    |   movel([-0.157173, -0.854007, -2.792927, -1.065455, 1.570796, 1.413623],accel_mss,speed_ms,0,blend_radius_m)
    |   movel([-0.155636, -0.852773, -2.793167, -1.066449, 1.570796, 1.415161],accel_mss,speed_ms,0,blend_radius_m)
    |   movel([-0.153982, -0.851875, -2.793341, -1.067172, 1.570796, 1.416814],accel_mss,speed_ms,0,blend_radius_m)
    |   movel([-0.150724, -0.850900, -2.793530, -1.067959, 1.570796, 1.420072],accel_mss,speed_ms,0,blend_radius_m)
    |   movel([-0.148143, -0.850668, -2.793575, -1.068146, 1.570796, 1.422653],accel_mss,speed_ms,0,blend_radius_m)
    |   movel([-0.149321, -0.848135, -2.794062, -1.070192, 1.570796, 1.421476],accel_mss,speed_ms,0,blend_radius_m)
    |   movel([-0.151025, -0.846251, -2.794422, -1.071716, 1.570796, 1.419772],accel_mss,speed_ms,0,blend_radius_m)
    |   movel([-0.155392, -0.843635, -2.794919, -1.073835, 1.570796, 1.415404],accel_mss,speed_ms,0,blend_radius_m)
    |   movel([-0.159988, -0.841179, -2.795382, -1.075828, 1.570796, 1.410808],accel_mss,speed_ms,0,blend_radius_m)
    |   movel([-0.161984, -0.839490, -2.795698, -1.077201, 1.570796, 1.408813],accel_mss,speed_ms,0,blend_radius_m)
    |   movel([-0.163557, -0.837206, -2.796124, -1.079060, 1.570796, 1.407239],accel_mss,speed_ms,0,blend_radius_m)
    |   movel([-0.164261, -0.835458, -2.796447, -1.080484, 1.570796, 1.406535],accel_mss,speed_ms,0,blend_radius_m)
    |   movel([-0.164602, -0.833827, -2.796748, -1.081815, 1.570796, 1.406195],accel_mss,speed_ms,0,blend_radius_m)
    |   movel([-0.164612, -0.832318, -2.797024, -1.083047, 1.570796, 1.406184],accel_mss,speed_ms,0,blend_radius_m)
    |   movel([-0.164323, -0.830942, -2.797275, -1.084171, 1.570796, 1.406473],accel_mss,speed_ms,0,blend_radius_m)
    |   movel([-0.163779, -0.829715, -2.797499, -1.085176, 1.570796, 1.407017],accel_mss,speed_ms,0,blend_radius_m)
    |   movel([-0.163009, -0.828631, -2.797695, -1.086063, 1.570796, 1.407787],accel_mss,speed_ms,0,blend_radius_m)
    |   movel([-0.162059, -0.827711, -2.797861, -1.086817, 1.570796, 1.408737],accel_mss,speed_ms,0,blend_radius_m)
    |   movel([-0.160956, -0.826959, -2.797997, -1.087433, 1.570796, 1.409840],accel_mss,speed_ms,0,blend_radius_m)
    |   movel([-0.159743, -0.826388, -2.798099, -1.087901, 1.570796, 1.411053],accel_mss,speed_ms,0,blend_radius_m)
    |   movel([-0.158463, -0.826010, -2.798167, -1.088211, 1.570796, 1.412333],accel_mss,speed_ms,0,blend_radius_m)
    |   movel([-0.155834, -0.825858, -2.798195, -1.088336, 1.570796, 1.414963],accel_mss,speed_ms,0,blend_radius_m)
    |   movel([-0.153372, -0.826573, -2.798066, -1.087750, 1.570796, 1.417424],accel_mss,speed_ms,0,blend_radius_m)
    |   movel([-0.151377, -0.828225, -2.797768, -1.086396, 1.570796, 1.419420],accel_mss,speed_ms,0,blend_radius_m)
    |   movel([-0.151142, -0.825056, -2.798338, -1.088994, 1.570796, 1.419654],accel_mss,speed_ms,0,blend_radius_m)
    |   movel([-0.151297, -0.822338, -2.798823, -1.091228, 1.570796, 1.419499],accel_mss,speed_ms,0,blend_radius_m)
    |   movel([-0.151760, -0.819974, -2.799241, -1.093173, 1.570796, 1.419036],accel_mss,speed_ms,0,blend_radius_m)
    |   movel([-0.154101, -0.813819, -2.800316, -1.098253, 1.570796, 1.416695],accel_mss,speed_ms,0,blend_radius_m)
    |   movel([-0.155566, -0.809336, -2.801087, -1.101966, 1.570796, 1.415230],accel_mss,speed_ms,0,blend_radius_m)
    |   movel([-0.155893, -0.807231, -2.801445, -1.103713, 1.570796, 1.414904],accel_mss,speed_ms,0,blend_radius_m)
    |   movel([-0.155922, -0.805199, -2.801789, -1.105401, 1.570796, 1.414875],accel_mss,speed_ms,0,blend_radius_m)
    |   movel([-0.155690, -0.803274, -2.802112, -1.107003, 1.570796, 1.415106],accel_mss,speed_ms,0,blend_radius_m)
    |   movel([-0.155226, -0.801477, -2.802413, -1.108500, 1.570796, 1.415570],accel_mss,speed_ms,0,blend_radius_m)
    |   movel([-0.154569, -0.799836, -2.802685, -1.109868, 1.570796, 1.416227],accel_mss,speed_ms,0,blend_radius_m)
    |   movel([-0.153748, -0.798375, -2.802927, -1.111087, 1.570796, 1.417049],accel_mss,speed_ms,0,blend_radius_m)
    |   movel([-0.152797, -0.797121, -2.803133, -1.112135, 1.570796, 1.417999],accel_mss,speed_ms,0,blend_radius_m)
    |   movel([-0.151752, -0.796103, -2.803301, -1.112985, 1.570796, 1.419044],accel_mss,speed_ms,0,blend_radius_m)
    |   movel([-0.150649, -0.795350, -2.803424, -1.113616, 1.570796, 1.420147],accel_mss,speed_ms,0,blend_radius_m)
    |   movel([-0.149524, -0.794885, -2.803500, -1.114004, 1.570796, 1.421272],accel_mss,speed_ms,0,blend_radius_m)
    |   movel([-0.148407, -0.794733, -2.803525, -1.114131, 1.570796, 1.422389],accel_mss,speed_ms,0,blend_radius_m)
    |   movel([-0.147335, -0.794925, -2.803493, -1.113970, 1.570796, 1.423462],accel_mss,speed_ms,0,blend_radius_m)
    |   movel([-0.146348, -0.795490, -2.803401, -1.113498, 1.570796, 1.424449],accel_mss,speed_ms,0,blend_radius_m)
    |   movel([-0.145476, -0.796449, -2.803244, -1.112696, 1.570796, 1.425320],accel_mss,speed_ms,0,blend_radius_m)
    |   movel([-0.144756, -0.797829, -2.803017, -1.111543, 1.570796, 1.426040],accel_mss,speed_ms,0,blend_radius_m)
    |   movel([-0.144218, -0.799645, -2.802717, -1.110027, 1.570796, 1.426578],accel_mss,speed_ms,0,blend_radius_m)
    |   movel([-0.142768, -0.796226, -2.803280, -1.112882, 1.570796, 1.428028],accel_mss,speed_ms,0,blend_radius_m)
    |   movel([-0.141654, -0.792950, -2.803815, -1.115625, 1.570796, 1.429142],accel_mss,speed_ms,0,blend_radius_m)
    |   movel([-0.140811, -0.789788, -2.804325, -1.118275, 1.570796, 1.429985],accel_mss,speed_ms,0,blend_radius_m)
    |   movel([-0.140168, -0.786710, -2.804817, -1.120861, 1.570796, 1.430628],accel_mss,speed_ms,0,blend_radius_m)
    |   movel([-0.138139, -0.774609, -2.806707, -1.131074, 1.570796, 1.432657],accel_mss,speed_ms,0,blend_radius_m)
    |   movel([-0.137268, -0.770063, -2.807398, -1.134928, 1.570796, 1.433528],accel_mss,speed_ms,0,blend_radius_m)
    |   movel([-0.135786, -0.764437, -2.808239, -1.139713, 1.570796, 1.435010],accel_mss,speed_ms,0,blend_radius_m)
    |   movel([-0.134635, -0.761547, -2.808665, -1.142177, 1.570796, 1.436162],accel_mss,speed_ms,0,blend_radius_m)
    |   movel([-0.133113, -0.758786, -2.809068, -1.144534, 1.570796, 1.437684],accel_mss,speed_ms,0,blend_radius_m)
    |   movel([-0.132184, -0.757494, -2.809256, -1.145639, 1.570796, 1.438613],accel_mss,speed_ms,0,blend_radius_m)
    |   movel([-0.129965, -0.755171, -2.809591, -1.147627, 1.570796, 1.440832],accel_mss,speed_ms,0,blend_radius_m)
    |   movel([-0.128651, -0.754181, -2.809733, -1.148475, 1.570796, 1.442146],accel_mss,speed_ms,0,blend_radius_m)
    |   movel([-0.127337, -0.753612, -2.809815, -1.148962, 1.570796, 1.443459],accel_mss,speed_ms,0,blend_radius_m)
    |   movel([-0.126342, -0.753754, -2.809794, -1.148841, 1.570796, 1.444454],accel_mss,speed_ms,0,blend_radius_m)
    |   movel([-0.125121, -0.755288, -2.809574, -1.147527, 1.570796, 1.445675],accel_mss,speed_ms,0,blend_radius_m)
    |   movel([-0.124184, -0.758153, -2.809161, -1.145076, 1.570796, 1.446612],accel_mss,speed_ms,0,blend_radius_m)
    |   movel([-0.123601, -0.761345, -2.808695, -1.142350, 1.570796, 1.447196],accel_mss,speed_ms,0,blend_radius_m)
    |   movel([-0.121151, -0.756396, -2.809415, -1.146579, 1.570796, 1.449645],accel_mss,speed_ms,0,blend_radius_m)
    |   movel([-0.118326, -0.751367, -2.810134, -1.150887, 1.570796, 1.452470],accel_mss,speed_ms,0,blend_radius_m)
    |   movel([-0.115181, -0.746327, -2.810844, -1.155218, 1.570796, 1.455615],accel_mss,speed_ms,0,blend_radius_m)
    |   movel([-0.111786, -0.741349, -2.811533, -1.159508, 1.570796, 1.459011],accel_mss,speed_ms,0,blend_radius_m)
    |   movel([-0.104952, -0.731339, -2.812883, -1.168167, 1.570796, 1.465845],accel_mss,speed_ms,0,blend_radius_m)
    |   movel([-0.102905, -0.728573, -2.813248, -1.170568, 1.570796, 1.467892],accel_mss,speed_ms,0,blend_radius_m)
    |   movel([-0.100882, -0.726090, -2.813573, -1.172726, 1.570796, 1.469915],accel_mss,speed_ms,0,blend_radius_m)
    |   movel([-0.098956, -0.724081, -2.813833, -1.174475, 1.570796, 1.471840],accel_mss,speed_ms,0,blend_radius_m)
    |   movel([-0.097220, -0.722741, -2.814006, -1.175641, 1.570796, 1.473576],accel_mss,speed_ms,0,blend_radius_m)
    |   movel([-0.095733, -0.722296, -2.814064, -1.176030, 1.570796, 1.475063],accel_mss,speed_ms,0,blend_radius_m)
    |   movel([-0.094670, -0.722789, -2.814000, -1.175600, 1.570796, 1.476126],accel_mss,speed_ms,0,blend_radius_m)
    |   movel([-0.094003, -0.724018, -2.813842, -1.174529, 1.570796, 1.476793],accel_mss,speed_ms,0,blend_radius_m)
    |   movel([-0.093720, -0.725788, -2.813612, -1.172989, 1.570796, 1.477077],accel_mss,speed_ms,0,blend_radius_m)
    |   movel([-0.093794, -0.727894, -2.813337, -1.171158, 1.570796, 1.477002],accel_mss,speed_ms,0,blend_radius_m)
    |   movel([-0.094201, -0.730131, -2.813043, -1.169215, 1.570796, 1.476595],accel_mss,speed_ms,0,blend_radius_m)
    |   movel([-0.094921, -0.732302, -2.812755, -1.167332, 1.570796, 1.475876],accel_mss,speed_ms,0,blend_radius_m)
    |   movel([-0.095934, -0.734211, -2.812500, -1.165677, 1.570796, 1.474862],accel_mss,speed_ms,0,blend_radius_m)
    |   movel([-0.089576, -0.725324, -2.813672, -1.173393, 1.570796, 1.481220],accel_mss,speed_ms,0,blend_radius_m)
    |   movel([-0.086162, -0.720979, -2.814232, -1.177177, 1.570796, 1.484634],accel_mss,speed_ms,0,blend_radius_m)
    |   movel([-0.082605, -0.716751, -2.814769, -1.180869, 1.570796, 1.488191],accel_mss,speed_ms,0,blend_radius_m)
    |   movel([-0.078927, -0.712679, -2.815278, -1.184431, 1.570796, 1.491869],accel_mss,speed_ms,0,blend_radius_m)
    |   movel([-0.075137, -0.708803, -2.815756, -1.187829, 1.570796, 1.495659],accel_mss,speed_ms,0,blend_radius_m)
    |   movel([-0.071252, -0.705165, -2.816199, -1.191025, 1.570796, 1.499544],accel_mss,speed_ms,0,blend_radius_m)
    |   movel([-0.067291, -0.701802, -2.816603, -1.193984, 1.570796, 1.503506],accel_mss,speed_ms,0,blend_radius_m)
    |   movel([-0.064593, -0.700056, -2.816811, -1.195522, 1.570796, 1.506203],accel_mss,speed_ms,0,blend_radius_m)
    |   movel([-0.061701, -0.698911, -2.816946, -1.196532, 1.570796, 1.509095],accel_mss,speed_ms,0,blend_radius_m)
    |   movel([-0.060444, -0.698737, -2.816967, -1.196685, 1.570796, 1.510352],accel_mss,speed_ms,0,blend_radius_m)
    |   movel([-0.059448, -0.698913, -2.816946, -1.196530, 1.570796, 1.511348],accel_mss,speed_ms,0,blend_radius_m)
    |   movel([-0.058813, -0.699508, -2.816876, -1.196006, 1.570796, 1.511984],accel_mss,speed_ms,0,blend_radius_m)
    |   movel([-0.058648, -0.700593, -2.816747, -1.195049, 1.570796, 1.512148],accel_mss,speed_ms,0,blend_radius_m)
    |   movel([-0.059026, -0.702035, -2.816575, -1.193779, 1.570796, 1.511771],accel_mss,speed_ms,0,blend_radius_m)
    |   movel([-0.059804, -0.703666, -2.816380, -1.192343, 1.570796, 1.510992],accel_mss,speed_ms,0,blend_radius_m)
    |   movel([-0.062125, -0.707350, -2.815934, -1.189105, 1.570796, 1.508671],accel_mss,speed_ms,0,blend_radius_m)
    |   movel([-0.064902, -0.710819, -2.815509, -1.186061, 1.570796, 1.505895],accel_mss,speed_ms,0,blend_radius_m)
    |   movel([-0.067942, -0.714038, -2.815109, -1.183242, 1.570796, 1.502854],accel_mss,speed_ms,0,blend_radius_m)
    |   movel([-0.071057, -0.716970, -2.814741, -1.180677, 1.570796, 1.499740],accel_mss,speed_ms,0,blend_radius_m)
    |   movel([-0.067028, -0.715222, -2.814961, -1.182206, 1.570796, 1.503768],accel_mss,speed_ms,0,blend_radius_m)
    |   movel([-0.062835, -0.712992, -2.815240, -1.184158, 1.570796, 1.507961],accel_mss,speed_ms,0,blend_radius_m)
    |   movel([-0.058521, -0.710309, -2.815572, -1.186509, 1.570796, 1.512275],accel_mss,speed_ms,0,blend_radius_m)
    |   movel([-0.054124, -0.707195, -2.815953, -1.189242, 1.570796, 1.516672],accel_mss,speed_ms,0,blend_radius_m)
    |   movel([-0.050646, -0.704373, -2.816295, -1.191722, 1.570796, 1.520151],accel_mss,speed_ms,0,blend_radius_m)
    |   movel([-0.043815, -0.698292, -2.817019, -1.197078, 1.570796, 1.526981],accel_mss,speed_ms,0,blend_radius_m)
    |   movel([-0.040303, -0.695418, -2.817356, -1.199615, 1.570796, 1.530493],accel_mss,speed_ms,0,blend_radius_m)
    |   movel([-0.036299, -0.692430, -2.817703, -1.202257, 1.570796, 1.534498],accel_mss,speed_ms,0,blend_radius_m)
    |   movel([-0.029550, -0.687751, -2.818237, -1.206401, 1.570796, 1.541246],accel_mss,speed_ms,0,blend_radius_m)
    |   movel([-0.026322, -0.685794, -2.818458, -1.208137, 1.570796, 1.544475],accel_mss,speed_ms,0,blend_radius_m)
    |   movel([-0.023824, -0.684639, -2.818588, -1.209162, 1.570796, 1.546972],accel_mss,speed_ms,0,blend_radius_m)
    |   movel([-0.022997, -0.684488, -2.818605, -1.209296, 1.570796, 1.547799],accel_mss,speed_ms,0,blend_radius_m)
    |   movel([-0.022536, -0.684694, -2.818582, -1.209113, 1.570796, 1.548260],accel_mss,speed_ms,0,blend_radius_m)
    |   movel([-0.022492, -0.685295, -2.818514, -1.208579, 1.570796, 1.548305],accel_mss,speed_ms,0,blend_radius_m)
    |   movel([-0.022929, -0.686348, -2.818396, -1.207645, 1.570796, 1.547867],accel_mss,speed_ms,0,blend_radius_m)
    |   movel([-0.024592, -0.689011, -2.818094, -1.205283, 1.570796, 1.546204],accel_mss,speed_ms,0,blend_radius_m)
    |   movel([-0.026746, -0.691820, -2.817773, -1.202796, 1.570796, 1.544050],accel_mss,speed_ms,0,blend_radius_m)
    |   movel([-0.029251, -0.694704, -2.817439, -1.200246, 1.570796, 1.541546],accel_mss,speed_ms,0,blend_radius_m)
    |   movel([-0.031954, -0.697567, -2.817105, -1.197717, 1.570796, 1.538842],accel_mss,speed_ms,0,blend_radius_m)
    |   movel([-0.037413, -0.702922, -2.816469, -1.192998, 1.570796, 1.533384],accel_mss,speed_ms,0,blend_radius_m)
    |   movel([-0.041996, -0.707237, -2.815948, -1.189204, 1.570796, 1.528800],accel_mss,speed_ms,0,blend_radius_m)
    |   movel([-0.039684, -0.706721, -2.816010, -1.189657, 1.570796, 1.531113],accel_mss,speed_ms,0,blend_radius_m)
    |   movel([-0.037246, -0.705917, -2.816108, -1.190364, 1.570796, 1.533551],accel_mss,speed_ms,0,blend_radius_m)
    |   movel([-0.032075, -0.703597, -2.816388, -1.192404, 1.570796, 1.538721],accel_mss,speed_ms,0,blend_radius_m)
    |   movel([-0.026629, -0.700547, -2.816752, -1.195089, 1.570796, 1.544167],accel_mss,speed_ms,0,blend_radius_m)
    |   movel([-0.021050, -0.697047, -2.817166, -1.198176, 1.570796, 1.549746],accel_mss,speed_ms,0,blend_radius_m)
    |   movel([-0.016407, -0.693865, -2.817537, -1.200987, 1.570796, 1.554390],accel_mss,speed_ms,0,blend_radius_m)
    |   movel([-0.002304, -0.683687, -2.818694, -1.210008, 1.570796, 1.568493],accel_mss,speed_ms,0,blend_radius_m)
    |   movel([0.000307, -0.682237, -2.818856, -1.211296, 1.570796, 1.571103],accel_mss,speed_ms,0,blend_radius_m)
    |   movel([0.002343, -0.681707, -2.818914, -1.211768, 1.570796, 1.573139],accel_mss,speed_ms,0,blend_radius_m)
    |   movel([0.002760, -0.682018, -2.818880, -1.211491, 1.570796, 1.573556],accel_mss,speed_ms,0,blend_radius_m)
    |   movel([0.002568, -0.682838, -2.818789, -1.210762, 1.570796, 1.573364],accel_mss,speed_ms,0,blend_radius_m)
    |   movel([0.001613, -0.684258, -2.818631, -1.209501, 1.570796, 1.572410],accel_mss,speed_ms,0,blend_radius_m)
    |   movel([-0.000256, -0.686365, -2.818394, -1.207630, 1.570796, 1.570541],accel_mss,speed_ms,0,blend_radius_m)
    |   movel([-0.003382, -0.689438, -2.818046, -1.204905, 1.570796, 1.567415],accel_mss,speed_ms,0,blend_radius_m)
    |   movel([-0.006983, -0.692611, -2.817682, -1.202096, 1.570796, 1.563814],accel_mss,speed_ms,0,blend_radius_m)
    |   movel([-0.010526, -0.695305, -2.817369, -1.199714, 1.570796, 1.560271],accel_mss,speed_ms,0,blend_radius_m)
    |   movel([-0.012112, -0.696296, -2.817254, -1.198839, 1.570796, 1.558684],accel_mss,speed_ms,0,blend_radius_m)
    |   movel([-0.013481, -0.696943, -2.817178, -1.198268, 1.570796, 1.557315],accel_mss,speed_ms,0,blend_radius_m)
    |   movel([-0.008162, -0.696506, -2.817229, -1.198654, 1.570796, 1.562634],accel_mss,speed_ms,0,blend_radius_m)
    |   movel([-0.002460, -0.695324, -2.817367, -1.199698, 1.570796, 1.568336],accel_mss,speed_ms,0,blend_radius_m)
    |   movel([0.003547, -0.693539, -2.817574, -1.201275, 1.570796, 1.574343],accel_mss,speed_ms,0,blend_radius_m)
    |   movel([0.009790, -0.691297, -2.817833, -1.203259, 1.570796, 1.580586],accel_mss,speed_ms,0,blend_radius_m)
    |   movel([0.022658, -0.686000, -2.818435, -1.207954, 1.570796, 1.593454],accel_mss,speed_ms,0,blend_radius_m)
    |   movel([0.035476, -0.680608, -2.819036, -1.212745, 1.570796, 1.606273],accel_mss,speed_ms,0,blend_radius_m)
    |   movel([0.037595, -0.680073, -2.819095, -1.213222, 1.570796, 1.608391],accel_mss,speed_ms,0,blend_radius_m)
    |   movel([0.038280, -0.680335, -2.819066, -1.212988, 1.570796, 1.609077],accel_mss,speed_ms,0,blend_radius_m)
    |   movel([0.038454, -0.681179, -2.818973, -1.212237, 1.570796, 1.609251],accel_mss,speed_ms,0,blend_radius_m)
    |   movel([0.038045, -0.682450, -2.818832, -1.211107, 1.570796, 1.608841],accel_mss,speed_ms,0,blend_radius_m)
    |   movel([0.035891, -0.686011, -2.818434, -1.207944, 1.570796, 1.606687],accel_mss,speed_ms,0,blend_radius_m)
    |   movel([0.034360, -0.688066, -2.818202, -1.206121, 1.570796, 1.605157],accel_mss,speed_ms,0,blend_radius_m)
    |   movel([0.030931, -0.691910, -2.817763, -1.202716, 1.570796, 1.601727],accel_mss,speed_ms,0,blend_radius_m)
    |   movel([0.027173, -0.695360, -2.817363, -1.199666, 1.570796, 1.597970],accel_mss,speed_ms,0,blend_radius_m)
    |   movel([0.023244, -0.698409, -2.817005, -1.196974, 1.570796, 1.594040],accel_mss,speed_ms,0,blend_radius_m)
    |   movel([0.019315, -0.701027, -2.816695, -1.194667, 1.570796, 1.590111],accel_mss,speed_ms,0,blend_radius_m)
    |   movel([0.015548, -0.703199, -2.816436, -1.192754, 1.570796, 1.586344],accel_mss,speed_ms,0,blend_radius_m)
    |   movel([0.012105, -0.704898, -2.816231, -1.191260, 1.570796, 1.582901],accel_mss,speed_ms,0,blend_radius_m)
    |   movel([0.009158, -0.706089, -2.816087, -1.190213, 1.570796, 1.579955],accel_mss,speed_ms,0,blend_radius_m)
    |   movel([0.009122, -0.706976, -2.815979, -1.189433, 1.570796, 1.579918],accel_mss,speed_ms,0,blend_radius_m)
    |   movel([0.009634, -0.707378, -2.815930, -1.189081, 1.570796, 1.580430],accel_mss,speed_ms,0,blend_radius_m)
    |   movel([0.011224, -0.707724, -2.815888, -1.188777, 1.570796, 1.582020],accel_mss,speed_ms,0,blend_radius_m)
    |   movel([0.013030, -0.707717, -2.815889, -1.188783, 1.570796, 1.583826],accel_mss,speed_ms,0,blend_radius_m)
    |   movel([0.017003, -0.707079, -2.815967, -1.189343, 1.570796, 1.587799],accel_mss,speed_ms,0,blend_radius_m)
    |   movel([0.024091, -0.705495, -2.816159, -1.190735, 1.570796, 1.594887],accel_mss,speed_ms,0,blend_radius_m)
    |   movel([0.031302, -0.703602, -2.816387, -1.192399, 1.570796, 1.602098],accel_mss,speed_ms,0,blend_radius_m)
    |   movel([0.046101, -0.699018, -2.816934, -1.196438, 1.570796, 1.616897],accel_mss,speed_ms,0,blend_radius_m)
    |   movel([0.050206, -0.697835, -2.817073, -1.197481, 1.570796, 1.621002],accel_mss,speed_ms,0,blend_radius_m)
    |   movel([0.052798, -0.697331, -2.817132, -1.197926, 1.570796, 1.623594],accel_mss,speed_ms,0,blend_radius_m)
    |   movel([0.055274, -0.697154, -2.817153, -1.198082, 1.570796, 1.626070],accel_mss,speed_ms,0,blend_radius_m)
    |   movel([0.057259, -0.697513, -2.817111, -1.197765, 1.570796, 1.628055],accel_mss,speed_ms,0,blend_radius_m)
    |   movel([0.058392, -0.698596, -2.816983, -1.196809, 1.570796, 1.629188],accel_mss,speed_ms,0,blend_radius_m)
    |   movel([0.058534, -0.699464, -2.816881, -1.196044, 1.570796, 1.629331],accel_mss,speed_ms,0,blend_radius_m)
    |   movel([0.058333, -0.700583, -2.816748, -1.195058, 1.570796, 1.629130],accel_mss,speed_ms,0,blend_radius_m)
    |   movel([0.057737, -0.701985, -2.816581, -1.193823, 1.570796, 1.628533],accel_mss,speed_ms,0,blend_radius_m)
    |   movel([0.056715, -0.703679, -2.816378, -1.192332, 1.570796, 1.627511],accel_mss,speed_ms,0,blend_radius_m)
    |   movel([0.055222, -0.705253, -2.816188, -1.190947, 1.570796, 1.626018],accel_mss,speed_ms,0,blend_radius_m)
    |   movel([0.053193, -0.706766, -2.816005, -1.189618, 1.570796, 1.623989],accel_mss,speed_ms,0,blend_radius_m)
    |   movel([0.042343, -0.713656, -2.815157, -1.183576, 1.570796, 1.613139],accel_mss,speed_ms,0,blend_radius_m)
    |   movel([0.038709, -0.715494, -2.814927, -1.181968, 1.570796, 1.609506],accel_mss,speed_ms,0,blend_radius_m)
    |   movel([0.037151, -0.716027, -2.814860, -1.181502, 1.570796, 1.607947],accel_mss,speed_ms,0,blend_radius_m)
    |   movel([0.035867, -0.716186, -2.814840, -1.181363, 1.570796, 1.606663],accel_mss,speed_ms,0,blend_radius_m)
    |   movel([0.041190, -0.717593, -2.814663, -1.180133, 1.570796, 1.611986],accel_mss,speed_ms,0,blend_radius_m)
    |   movel([0.047112, -0.718032, -2.814607, -1.179749, 1.570796, 1.617908],accel_mss,speed_ms,0,blend_radius_m)
    |   movel([0.053494, -0.717683, -2.814651, -1.180054, 1.570796, 1.624290],accel_mss,speed_ms,0,blend_radius_m)
    |   movel([0.060203, -0.716712, -2.814774, -1.180903, 1.570796, 1.630999],accel_mss,speed_ms,0,blend_radius_m)
    |   movel([0.066007, -0.715025, -2.814986, -1.182378, 1.570796, 1.636803],accel_mss,speed_ms,0,blend_radius_m)
    |   movel([0.074325, -0.712783, -2.815265, -1.184340, 1.570796, 1.645121],accel_mss,speed_ms,0,blend_radius_m)
    |   movel([0.078086, -0.712239, -2.815333, -1.184817, 1.570796, 1.648883],accel_mss,speed_ms,0,blend_radius_m)
    |   movel([0.080879, -0.712477, -2.815303, -1.184608, 1.570796, 1.651675],accel_mss,speed_ms,0,blend_radius_m)
    |   movel([0.081744, -0.712983, -2.815241, -1.184166, 1.570796, 1.652541],accel_mss,speed_ms,0,blend_radius_m)
    |   movel([0.082165, -0.713793, -2.815140, -1.183456, 1.570796, 1.652962],accel_mss,speed_ms,0,blend_radius_m)
    |   movel([0.082079, -0.714949, -2.814995, -1.182444, 1.570796, 1.652876],accel_mss,speed_ms,0,blend_radius_m)
    |   movel([0.081432, -0.716473, -2.814804, -1.181112, 1.570796, 1.652228],accel_mss,speed_ms,0,blend_radius_m)
    |   movel([0.080447, -0.718044, -2.814606, -1.179739, 1.570796, 1.651243],accel_mss,speed_ms,0,blend_radius_m)
    |   movel([0.079310, -0.719549, -2.814415, -1.178425, 1.570796, 1.650106],accel_mss,speed_ms,0,blend_radius_m)
    |   movel([0.076800, -0.722361, -2.814055, -1.175972, 1.570796, 1.647596],accel_mss,speed_ms,0,blend_radius_m)
    |   movel([0.074028, -0.725144, -2.813696, -1.173549, 1.570796, 1.644824],accel_mss,speed_ms,0,blend_radius_m)
    |   movel([0.068413, -0.730106, -2.813046, -1.169236, 1.570796, 1.639210],accel_mss,speed_ms,0,blend_radius_m)
    |   movel([0.065604, -0.732263, -2.812760, -1.167365, 1.570796, 1.636400],accel_mss,speed_ms,0,blend_radius_m)
    |   movel([0.070716, -0.731447, -2.812869, -1.168073, 1.570796, 1.641512],accel_mss,speed_ms,0,blend_radius_m)
    |   movel([0.075992, -0.730228, -2.813030, -1.169131, 1.570796, 1.646788],accel_mss,speed_ms,0,blend_radius_m)
    |   movel([0.081419, -0.728656, -2.813237, -1.170496, 1.570796, 1.652215],accel_mss,speed_ms,0,blend_radius_m)
    |   movel([0.086983, -0.726764, -2.813485, -1.172140, 1.570796, 1.657779],accel_mss,speed_ms,0,blend_radius_m)
    |   movel([0.098455, -0.722201, -2.814076, -1.176112, 1.570796, 1.669251],accel_mss,speed_ms,0,blend_radius_m)
    |   movel([0.110292, -0.716861, -2.814755, -1.180773, 1.570796, 1.681088],accel_mss,speed_ms,0,blend_radius_m)
    |   movel([0.113392, -0.715791, -2.814890, -1.181708, 1.570796, 1.684188],accel_mss,speed_ms,0,blend_radius_m)
    |   movel([0.114491, -0.715953, -2.814870, -1.181567, 1.570796, 1.685287],accel_mss,speed_ms,0,blend_radius_m)
    |   movel([0.114930, -0.716934, -2.814746, -1.180709, 1.570796, 1.685727],accel_mss,speed_ms,0,blend_radius_m)
    |   movel([0.114784, -0.717962, -2.814616, -1.179811, 1.570796, 1.685580],accel_mss,speed_ms,0,blend_radius_m)
    |   movel([0.114349, -0.719125, -2.814469, -1.178795, 1.570796, 1.685146],accel_mss,speed_ms,0,blend_radius_m)
    |   movel([0.112744, -0.721791, -2.814128, -1.176470, 1.570796, 1.683540],accel_mss,speed_ms,0,blend_radius_m)
    |   movel([0.110406, -0.724719, -2.813751, -1.173919, 1.570796, 1.681202],accel_mss,speed_ms,0,blend_radius_m)
    |   movel([0.107619, -0.727723, -2.813360, -1.171306, 1.570796, 1.678415],accel_mss,speed_ms,0,blend_radius_m)
    |   movel([0.101837, -0.733162, -2.812641, -1.166586, 1.570796, 1.672633],accel_mss,speed_ms,0,blend_radius_m)
    |   movel([0.097629, -0.736554, -2.812185, -1.163650, 1.570796, 1.668425],accel_mss,speed_ms,0,blend_radius_m)
    |   movel([0.099987, -0.735760, -2.812292, -1.164336, 1.570796, 1.670784],accel_mss,speed_ms,0,blend_radius_m)
    |   movel([0.102438, -0.734691, -2.812436, -1.165262, 1.570796, 1.673234],accel_mss,speed_ms,0,blend_radius_m)
    |   movel([0.107559, -0.731813, -2.812820, -1.167756, 1.570796, 1.678355],accel_mss,speed_ms,0,blend_radius_m)
    |   movel([0.112892, -0.728037, -2.813318, -1.171034, 1.570796, 1.683688],accel_mss,speed_ms,0,blend_radius_m)
    |   movel([0.118336, -0.723500, -2.813908, -1.174980, 1.570796, 1.689132],accel_mss,speed_ms,0,blend_radius_m)
    |   movel([0.123794, -0.718309, -2.814572, -1.179508, 1.570796, 1.694590],accel_mss,speed_ms,0,blend_radius_m)
    |   movel([0.129160, -0.712605, -2.815288, -1.184497, 1.570796, 1.699957],accel_mss,speed_ms,0,blend_radius_m)
    |   movel([0.134328, -0.706502, -2.816037, -1.189850, 1.570796, 1.705125],accel_mss,speed_ms,0,blend_radius_m)
    |   movel([0.139190, -0.700141, -2.816801, -1.195448, 1.570796, 1.709986],accel_mss,speed_ms,0,blend_radius_m)
    |   movel([0.141342, -0.697297, -2.817136, -1.197956, 1.570796, 1.712138],accel_mss,speed_ms,0,blend_radius_m)
    |   movel([0.142493, -0.696050, -2.817282, -1.199057, 1.570796, 1.713289],accel_mss,speed_ms,0,blend_radius_m)
    |   movel([0.143679, -0.695077, -2.817396, -1.199916, 1.570796, 1.714475],accel_mss,speed_ms,0,blend_radius_m)
    |   movel([0.144887, -0.694523, -2.817460, -1.200405, 1.570796, 1.715683],accel_mss,speed_ms,0,blend_radius_m)
    |   movel([0.145893, -0.694447, -2.817469, -1.200473, 1.570796, 1.716690],accel_mss,speed_ms,0,blend_radius_m)
    |   movel([0.146954, -0.695110, -2.817392, -1.199887, 1.570796, 1.717750],accel_mss,speed_ms,0,blend_radius_m)
    |   movel([0.147451, -0.696599, -2.817218, -1.198572, 1.570796, 1.718248],accel_mss,speed_ms,0,blend_radius_m)
    |   movel([0.147486, -0.698706, -2.816970, -1.196713, 1.570796, 1.718282],accel_mss,speed_ms,0,blend_radius_m)
    |   movel([0.147161, -0.701238, -2.816670, -1.194481, 1.570796, 1.717957],accel_mss,speed_ms,0,blend_radius_m)
    |   movel([0.145830, -0.706758, -2.816006, -1.189625, 1.570796, 1.716626],accel_mss,speed_ms,0,blend_radius_m)
    |   movel([0.144266, -0.711579, -2.815415, -1.185395, 1.570796, 1.715062],accel_mss,speed_ms,0,blend_radius_m)
    |   movel([0.148453, -0.705402, -2.816170, -1.190817, 1.570796, 1.719250],accel_mss,speed_ms,0,blend_radius_m)
    |   movel([0.152248, -0.699119, -2.816922, -1.196348, 1.570796, 1.723045],accel_mss,speed_ms,0,blend_radius_m)
    |   movel([0.155623, -0.692793, -2.817661, -1.201935, 1.570796, 1.726419],accel_mss,speed_ms,0,blend_radius_m)
    |   movel([0.158554, -0.686512, -2.818378, -1.207500, 1.570796, 1.729350],accel_mss,speed_ms,0,blend_radius_m)
    |   movel([0.160997, -0.680357, -2.819064, -1.212969, 1.570796, 1.731793],accel_mss,speed_ms,0,blend_radius_m)
    |   movel([0.162938, -0.674397, -2.819712, -1.218279, 1.570796, 1.733734],accel_mss,speed_ms,0,blend_radius_m)
    |   movel([0.164327, -0.668739, -2.820315, -1.223335, 1.570796, 1.735123],accel_mss,speed_ms,0,blend_radius_m)
    |   movel([0.165138, -0.663459, -2.820865, -1.228066, 1.570796, 1.735934],accel_mss,speed_ms,0,blend_radius_m)
    |   movel([0.165317, -0.656807, -2.821541, -1.234041, 1.570796, 1.736113],accel_mss,speed_ms,0,blend_radius_m)
    |   movel([0.165687, -0.653114, -2.821909, -1.237367, 1.570796, 1.736484],accel_mss,speed_ms,0,blend_radius_m)
    |   movel([0.166123, -0.651214, -2.822096, -1.239079, 1.570796, 1.736919],accel_mss,speed_ms,0,blend_radius_m)
    |   movel([0.166789, -0.649298, -2.822283, -1.240808, 1.570796, 1.737585],accel_mss,speed_ms,0,blend_radius_m)
    |   movel([0.168341, -0.646127, -2.822589, -1.243672, 1.570796, 1.739137],accel_mss,speed_ms,0,blend_radius_m)
    |   movel([0.169767, -0.644163, -2.822777, -1.245449, 1.570796, 1.740563],accel_mss,speed_ms,0,blend_radius_m)
    |   movel([0.171087, -0.643150, -2.822873, -1.246366, 1.570796, 1.741883],accel_mss,speed_ms,0,blend_radius_m)
    |   movel([0.172312, -0.642832, -2.822903, -1.246653, 1.570796, 1.743108],accel_mss,speed_ms,0,blend_radius_m)
    |   movel([0.175518, -0.643515, -2.822839, -1.246036, 1.570796, 1.746314],accel_mss,speed_ms,0,blend_radius_m)
    |   movel([0.176484, -0.643421, -2.822847, -1.246120, 1.570796, 1.747280],accel_mss,speed_ms,0,blend_radius_m)
    |   movel([0.178697, -0.638716, -2.823289, -1.250383, 1.570796, 1.749494],accel_mss,speed_ms,0,blend_radius_m)
    |   movel([0.180593, -0.634065, -2.823718, -1.254607, 1.570796, 1.751389],accel_mss,speed_ms,0,blend_radius_m)
    |   movel([0.182183, -0.629486, -2.824131, -1.258772, 1.570796, 1.752980],accel_mss,speed_ms,0,blend_radius_m)
    |   movel([0.183484, -0.624991, -2.824528, -1.262869, 1.570796, 1.754280],accel_mss,speed_ms,0,blend_radius_m)
    |   movel([0.184496, -0.620610, -2.824908, -1.266871, 1.570796, 1.755292],accel_mss,speed_ms,0,blend_radius_m)
    |   movel([0.185235, -0.616352, -2.825270, -1.270768, 1.570796, 1.756031],accel_mss,speed_ms,0,blend_radius_m)
    |   movel([0.185961, -0.608264, -2.825938, -1.278187, 1.570796, 1.756757],accel_mss,speed_ms,0,blend_radius_m)
    |   movel([0.185749, -0.600887, -2.826525, -1.284977, 1.570796, 1.756546],accel_mss,speed_ms,0,blend_radius_m)
    |   movel([0.184726, -0.594338, -2.827029, -1.291022, 1.570796, 1.755523],accel_mss,speed_ms,0,blend_radius_m)
    |   movel([0.182987, -0.588769, -2.827445, -1.296176, 1.570796, 1.753783],accel_mss,speed_ms,0,blend_radius_m)
    |   movel([0.180673, -0.584283, -2.827771, -1.300335, 1.570796, 1.751470],accel_mss,speed_ms,0,blend_radius_m)
    |   speed_ms = 0.005
    |   movel([0.180673, -0.578816, -2.820911, -1.312663, 1.570796, 1.751470],accel_mss,speed_ms,0,blend_radius_m)
    |   speed_ms = 0.040
    |   movel([0.147045, -0.606212, -2.818803, -1.287374, 1.570796, 1.717842],accel_mss,speed_ms,0,blend_radius_m)
    |   speed_ms = 0.005
    |   movel([0.147045, -0.612154, -2.825620, -1.274615, 1.570796, 1.717842],accel_mss,speed_ms,0,blend_radius_m)
    |   speed_ms = 0.025
    |   movel([0.144295, -0.611885, -2.825642, -1.274862, 1.570796, 1.715092],accel_mss,speed_ms,0,blend_radius_m)
    |   movel([0.141059, -0.612581, -2.825584, -1.274224, 1.570796, 1.711855],accel_mss,speed_ms,0,blend_radius_m)
    |   movel([0.137432, -0.614098, -2.825459, -1.272832, 1.570796, 1.708228],accel_mss,speed_ms,0,blend_radius_m)
    |   movel([0.133525, -0.616279, -2.825276, -1.270834, 1.570796, 1.704322],accel_mss,speed_ms,0,blend_radius_m)
    |   movel([0.129441, -0.618974, -2.825048, -1.268368, 1.570796, 1.700237],accel_mss,speed_ms,0,blend_radius_m)
    |   movel([0.125275, -0.622032, -2.824786, -1.265572, 1.570796, 1.696071],accel_mss,speed_ms,0,blend_radius_m)
    |   movel([0.117100, -0.628639, -2.824206, -1.259544, 1.570796, 1.687896],accel_mss,speed_ms,0,blend_radius_m)
    |   speed_ms = 0.005
    |   movel([0.117100, -0.622425, -2.817419, -1.272545, 1.570796, 1.687896],accel_mss,speed_ms,0,blend_radius_m)
    |   speed_ms = 0.040
    |   movel([0.127695, -0.613108, -2.818227, -1.281054, 1.570796, 1.698492],accel_mss,speed_ms,0,blend_radius_m)
    |   speed_ms = 0.005
    |   movel([0.127695, -0.619167, -2.825031, -1.268191, 1.570796, 1.698492],accel_mss,speed_ms,0,blend_radius_m)
    |   speed_ms = 0.025
    |   movel([0.129450, -0.614059, -2.825462, -1.272868, 1.570796, 1.700246],accel_mss,speed_ms,0,blend_radius_m)
    |   movel([0.130751, -0.609325, -2.825852, -1.277212, 1.570796, 1.701548],accel_mss,speed_ms,0,blend_radius_m)
    |   movel([0.131606, -0.604959, -2.826203, -1.281226, 1.570796, 1.702402],accel_mss,speed_ms,0,blend_radius_m)
    |   movel([0.132031, -0.600944, -2.826521, -1.284924, 1.570796, 1.702827],accel_mss,speed_ms,0,blend_radius_m)
    |   movel([0.132052, -0.597259, -2.826806, -1.288324, 1.570796, 1.702849],accel_mss,speed_ms,0,blend_radius_m)
    |   movel([0.131684, -0.593889, -2.827063, -1.291437, 1.570796, 1.702480],accel_mss,speed_ms,0,blend_radius_m)
    |   movel([0.130945, -0.590817, -2.827293, -1.294279, 1.570796, 1.701741],accel_mss,speed_ms,0,blend_radius_m)
    |   movel([0.129858, -0.588023, -2.827500, -1.296867, 1.570796, 1.700654],accel_mss,speed_ms,0,blend_radius_m)
    |   movel([0.125627, -0.580948, -2.828009, -1.303432, 1.570796, 1.696423],accel_mss,speed_ms,0,blend_radius_m)
    |   movel([0.123803, -0.577346, -2.828261, -1.306782, 1.570796, 1.694599],accel_mss,speed_ms,0,blend_radius_m)
    |   movel([0.122580, -0.572615, -2.828585, -1.311190, 1.570796, 1.693377],accel_mss,speed_ms,0,blend_radius_m)
    |   movel([0.121897, -0.565868, -2.829032, -1.317488, 1.570796, 1.692693],accel_mss,speed_ms,0,blend_radius_m)
    |   movel([0.121921, -0.558454, -2.829505, -1.324430, 1.570796, 1.692717],accel_mss,speed_ms,0,blend_radius_m)
    |   movel([0.122901, -0.550231, -2.830005, -1.332153, 1.570796, 1.693698],accel_mss,speed_ms,0,blend_radius_m)
    |   movel([0.123828, -0.545771, -2.830266, -1.336352, 1.570796, 1.694624],accel_mss,speed_ms,0,blend_radius_m)
    |   movel([0.125095, -0.541054, -2.830535, -1.340800, 1.570796, 1.695892],accel_mss,speed_ms,0,blend_radius_m)
    |   movel([0.127797, -0.533334, -2.830957, -1.348098, 1.570796, 1.698594],accel_mss,speed_ms,0,blend_radius_m)
    |   movel([0.131353, -0.525355, -2.831371, -1.355663, 1.570796, 1.702149],accel_mss,speed_ms,0,blend_radius_m)
    |   movel([0.135724, -0.517175, -2.831772, -1.363442, 1.570796, 1.706520],accel_mss,speed_ms,0,blend_radius_m)
    |   movel([0.140867, -0.508859, -2.832156, -1.371374, 1.570796, 1.711663],accel_mss,speed_ms,0,blend_radius_m)
    |   movel([0.146727, -0.500491, -2.832518, -1.379381, 1.570796, 1.717523],accel_mss,speed_ms,0,blend_radius_m)
    |   movel([0.153260, -0.492142, -2.832854, -1.387393, 1.570796, 1.724056],accel_mss,speed_ms,0,blend_radius_m)
    |   movel([0.160410, -0.483888, -2.833164, -1.395337, 1.570796, 1.731207],accel_mss,speed_ms,0,blend_radius_m)
    |   movel([0.168108, -0.475828, -2.833444, -1.403118, 1.570796, 1.738904],accel_mss,speed_ms,0,blend_radius_m)
    |   movel([0.174111, -0.470061, -2.833630, -1.408698, 1.570796, 1.744908],accel_mss,speed_ms,0,blend_radius_m)
    |   movel([0.180217, -0.464629, -2.833795, -1.413964, 1.570796, 1.751014],accel_mss,speed_ms,0,blend_radius_m)
    |   movel([0.186360, -0.459584, -2.833940, -1.418865, 1.570796, 1.757156],accel_mss,speed_ms,0,blend_radius_m)
    |   movel([0.192492, -0.454944, -2.834066, -1.423379, 1.570796, 1.763288],accel_mss,speed_ms,0,blend_radius_m)
    |   movel([0.198543, -0.450773, -2.834172, -1.427444, 1.570796, 1.769339],accel_mss,speed_ms,0,blend_radius_m)
    |   movel([0.204454, -0.447101, -2.834262, -1.431027, 1.570796, 1.775250],accel_mss,speed_ms,0,blend_radius_m)
    |   movel([0.210158, -0.443971, -2.834334, -1.434084, 1.570796, 1.780954],accel_mss,speed_ms,0,blend_radius_m)
    |   movel([0.215594, -0.441425, -2.834390, -1.436574, 1.570796, 1.786390],accel_mss,speed_ms,0,blend_radius_m)
    |   movel([0.220696, -0.439502, -2.834432, -1.438455, 1.570796, 1.791492],accel_mss,speed_ms,0,blend_radius_m)
    |   movel([0.225414, -0.438230, -2.834458, -1.439700, 1.570796, 1.796210],accel_mss,speed_ms,0,blend_radius_m)
    |   movel([0.229681, -0.437651, -2.834470, -1.440268, 1.570796, 1.800477],accel_mss,speed_ms,0,blend_radius_m)
    |   movel([0.233444, -0.437793, -2.834467, -1.440129, 1.570796, 1.804240],accel_mss,speed_ms,0,blend_radius_m)
    |   movel([0.236651, -0.438680, -2.834449, -1.439261, 1.570796, 1.807447],accel_mss,speed_ms,0,blend_radius_m)
    |   movel([0.239236, -0.440352, -2.834413, -1.437623, 1.570796, 1.810033],accel_mss,speed_ms,0,blend_radius_m)
    |   movel([0.241164, -0.442817, -2.834360, -1.435212, 1.570796, 1.811960],accel_mss,speed_ms,0,blend_radius_m)
    |   movel([0.242388, -0.446104, -2.834285, -1.432000, 1.570796, 1.813185],accel_mss,speed_ms,0,blend_radius_m)
    |   movel([0.243113, -0.451276, -2.834160, -1.426954, 1.570796, 1.813909],accel_mss,speed_ms,0,blend_radius_m)
    |   movel([0.243193, -0.457064, -2.834009, -1.421315, 1.570796, 1.813989],accel_mss,speed_ms,0,blend_radius_m)
    |   movel([0.242762, -0.463326, -2.833834, -1.415230, 1.570796, 1.813559],accel_mss,speed_ms,0,blend_radius_m)
    |   movel([0.241979, -0.469883, -2.833636, -1.408870, 1.570796, 1.812775],accel_mss,speed_ms,0,blend_radius_m)
    |   movel([0.239586, -0.484655, -2.833136, -1.394598, 1.570796, 1.810383],accel_mss,speed_ms,0,blend_radius_m)
    |   movel([0.236542, -0.499913, -2.832542, -1.379934, 1.570796, 1.807339],accel_mss,speed_ms,0,blend_radius_m)
    |   movel([0.233030, -0.515493, -2.831852, -1.365044, 1.570796, 1.803826],accel_mss,speed_ms,0,blend_radius_m)
    |   movel([0.229223, -0.531216, -2.831069, -1.350104, 1.570796, 1.800019],accel_mss,speed_ms,0,blend_radius_m)
    |   movel([0.214200, -0.592712, -2.827152, -1.292525, 1.570796, 1.784997],accel_mss,speed_ms,0,blend_radius_m)
    |   movel([0.208188, -0.621558, -2.824826, -1.266004, 1.570796, 1.778984],accel_mss,speed_ms,0,blend_radius_m)
    |   movel([0.205706, -0.635455, -2.823591, -1.253343, 1.570796, 1.776502],accel_mss,speed_ms,0,blend_radius_m)
    |   movel([0.203697, -0.648880, -2.822323, -1.241185, 1.570796, 1.774493],accel_mss,speed_ms,0,blend_radius_m)
    |   movel([0.202238, -0.661775, -2.821038, -1.229576, 1.570796, 1.773035],accel_mss,speed_ms,0,blend_radius_m)
    |   movel([0.201412, -0.674064, -2.819748, -1.218576, 1.570796, 1.772208],accel_mss,speed_ms,0,blend_radius_m)
    |   movel([0.201282, -0.685699, -2.818469, -1.208221, 1.570796, 1.772078],accel_mss,speed_ms,0,blend_radius_m)
    |   movel([0.201935, -0.696615, -2.817216, -1.198558, 1.570796, 1.772731],accel_mss,speed_ms,0,blend_radius_m)
    |   movel([0.202500, -0.700580, -2.816748, -1.195060, 1.570796, 1.773296],accel_mss,speed_ms,0,blend_radius_m)
    |   movel([0.203584, -0.704026, -2.816336, -1.192027, 1.570796, 1.774380],accel_mss,speed_ms,0,blend_radius_m)
    |   movel([0.205463, -0.706475, -2.816040, -1.189873, 1.570796, 1.776260],accel_mss,speed_ms,0,blend_radius_m)
    |   movel([0.206790, -0.707176, -2.815955, -1.189258, 1.570796, 1.777587],accel_mss,speed_ms,0,blend_radius_m)
    |   movel([0.208428, -0.707443, -2.815923, -1.189023, 1.570796, 1.779225],accel_mss,speed_ms,0,blend_radius_m)
    |   speed_ms = 0.005
    |   movel([0.208428, -0.700045, -2.809298, -1.203046, 1.570796, 1.779225],accel_mss,speed_ms,0,blend_radius_m)
    |   speed_ms = 0.040
    |   movel([0.175669, -0.661052, -2.813693, -1.237644, 1.570796, 1.746465],accel_mss,speed_ms,0,blend_radius_m)
    |   speed_ms = 0.005
    |   movel([0.175669, -0.667879, -2.820405, -1.224105, 1.570796, 1.746465],accel_mss,speed_ms,0,blend_radius_m)
    |   speed_ms = 0.025
    |   movel([0.174359, -0.669978, -2.820184, -1.222227, 1.570796, 1.745156],accel_mss,speed_ms,0,blend_radius_m)
    |   movel([0.173356, -0.672109, -2.819958, -1.220323, 1.570796, 1.744153],accel_mss,speed_ms,0,blend_radius_m)
    |   movel([0.172639, -0.674239, -2.819729, -1.218420, 1.570796, 1.743436],accel_mss,speed_ms,0,blend_radius_m)
    |   movel([0.172156, -0.676387, -2.819497, -1.216504, 1.570796, 1.742952],accel_mss,speed_ms,0,blend_radius_m)
    |   movel([0.171785, -0.680659, -2.819030, -1.212700, 1.570796, 1.742581],accel_mss,speed_ms,0,blend_radius_m)
    |   movel([0.171963, -0.684857, -2.818564, -1.208969, 1.570796, 1.742760],accel_mss,speed_ms,0,blend_radius_m)
    |   movel([0.173142, -0.696316, -2.817251, -1.198822, 1.570796, 1.743938],accel_mss,speed_ms,0,blend_radius_m)
    |   movel([0.172873, -0.699513, -2.816875, -1.196001, 1.570796, 1.743669],accel_mss,speed_ms,0,blend_radius_m)
    |   movel([0.172311, -0.701120, -2.816684, -1.194585, 1.570796, 1.743108],accel_mss,speed_ms,0,blend_radius_m)
    |   movel([0.171360, -0.702511, -2.816518, -1.193359, 1.570796, 1.742157],accel_mss,speed_ms,0,blend_radius_m)
    |   movel([0.170465, -0.703358, -2.816417, -1.192614, 1.570796, 1.741262],accel_mss,speed_ms,0,blend_radius_m)
    |   movel([0.169625, -0.703720, -2.816373, -1.192296, 1.570796, 1.740421],accel_mss,speed_ms,0,blend_radius_m)
    |   movel([0.168835, -0.703668, -2.816379, -1.192342, 1.570796, 1.739631],accel_mss,speed_ms,0,blend_radius_m)
    |   movel([0.167422, -0.702532, -2.816516, -1.193341, 1.570796, 1.738218],accel_mss,speed_ms,0,blend_radius_m)
    |   movel([0.166234, -0.700439, -2.816765, -1.195185, 1.570796, 1.737030],accel_mss,speed_ms,0,blend_radius_m)
    |   movel([0.164582, -0.695278, -2.817372, -1.199738, 1.570796, 1.735378],accel_mss,speed_ms,0,blend_radius_m)
    |   movel([0.164030, -0.691990, -2.817753, -1.202646, 1.570796, 1.734826],accel_mss,speed_ms,0,blend_radius_m)
    |   movel([0.162204, -0.697996, -2.817054, -1.197339, 1.570796, 1.733001],accel_mss,speed_ms,0,blend_radius_m)
    |   movel([0.161124, -0.703567, -2.816392, -1.192430, 1.570796, 1.731920],accel_mss,speed_ms,0,blend_radius_m)
    |   movel([0.160676, -0.708742, -2.815764, -1.187883, 1.570796, 1.731472],accel_mss,speed_ms,0,blend_radius_m)
    |   movel([0.160765, -0.713527, -2.815173, -1.183689, 1.570796, 1.731562],accel_mss,speed_ms,0,blend_radius_m)
    |   movel([0.161279, -0.717966, -2.814616, -1.179807, 1.570796, 1.732075],accel_mss,speed_ms,0,blend_radius_m)
    |   movel([0.162133, -0.722059, -2.814094, -1.176236, 1.570796, 1.732929],accel_mss,speed_ms,0,blend_radius_m)
    |   movel([0.164443, -0.729307, -2.813151, -1.169930, 1.570796, 1.735239],accel_mss,speed_ms,0,blend_radius_m)
    |   movel([0.164488, -0.731052, -2.812921, -1.168416, 1.570796, 1.735284],accel_mss,speed_ms,0,blend_radius_m)
    |   movel([0.164087, -0.732059, -2.812787, -1.167543, 1.570796, 1.734883],accel_mss,speed_ms,0,blend_radius_m)
    |   movel([0.163334, -0.732926, -2.812672, -1.166791, 1.570796, 1.734130],accel_mss,speed_ms,0,blend_radius_m)
    |   movel([0.162378, -0.733363, -2.812614, -1.166412, 1.570796, 1.733174],accel_mss,speed_ms,0,blend_radius_m)
    |   movel([0.160324, -0.733609, -2.812581, -1.166199, 1.570796, 1.731121],accel_mss,speed_ms,0,blend_radius_m)
    |   movel([0.158612, -0.733307, -2.812621, -1.166461, 1.570796, 1.729408],accel_mss,speed_ms,0,blend_radius_m)
    |   movel([0.157197, -0.732541, -2.812723, -1.167125, 1.570796, 1.727993],accel_mss,speed_ms,0,blend_radius_m)
    |   movel([0.156057, -0.731366, -2.812880, -1.168144, 1.570796, 1.726853],accel_mss,speed_ms,0,blend_radius_m)
    |   movel([0.154474, -0.728099, -2.813310, -1.170980, 1.570796, 1.725270],accel_mss,speed_ms,0,blend_radius_m)
    |   movel([0.153620, -0.724072, -2.813835, -1.174482, 1.570796, 1.724417],accel_mss,speed_ms,0,blend_radius_m)
    |   movel([0.152734, -0.733420, -2.812606, -1.166363, 1.570796, 1.723531],accel_mss,speed_ms,0,blend_radius_m)
    |   movel([0.152749, -0.737685, -2.812032, -1.162672, 1.570796, 1.723545],accel_mss,speed_ms,0,blend_radius_m)
    |   movel([0.153326, -0.741490, -2.811513, -1.159386, 1.570796, 1.724123],accel_mss,speed_ms,0,blend_radius_m)
    |   movel([0.154543, -0.744124, -2.811150, -1.157115, 1.570796, 1.725340],accel_mss,speed_ms,0,blend_radius_m)
    |   movel([0.157840, -0.748112, -2.810594, -1.153683, 1.570796, 1.728637],accel_mss,speed_ms,0,blend_radius_m)
    |   movel([0.158957, -0.750728, -2.810225, -1.151436, 1.570796, 1.729754],accel_mss,speed_ms,0,blend_radius_m)
    |   movel([0.159040, -0.751388, -2.810131, -1.150869, 1.570796, 1.729837],accel_mss,speed_ms,0,blend_radius_m)
    |   movel([0.158835, -0.752228, -2.810012, -1.150149, 1.570796, 1.729631],accel_mss,speed_ms,0,blend_radius_m)
    |   movel([0.158181, -0.753138, -2.809882, -1.149369, 1.570796, 1.728977],accel_mss,speed_ms,0,blend_radius_m)
    |   movel([0.157098, -0.754023, -2.809756, -1.148610, 1.570796, 1.727895],accel_mss,speed_ms,0,blend_radius_m)
    |   movel([0.154213, -0.755638, -2.809524, -1.147227, 1.570796, 1.725009],accel_mss,speed_ms,0,blend_radius_m)
    |   movel([0.149460, -0.757553, -2.809247, -1.145588, 1.570796, 1.720256],accel_mss,speed_ms,0,blend_radius_m)
    |   movel([0.150003, -0.759871, -2.808910, -1.143607, 1.570796, 1.720799],accel_mss,speed_ms,0,blend_radius_m)
    |   movel([0.150887, -0.762343, -2.808548, -1.141498, 1.570796, 1.721683],accel_mss,speed_ms,0,blend_radius_m)
    |   movel([0.152214, -0.764783, -2.808188, -1.139418, 1.570796, 1.723011],accel_mss,speed_ms,0,blend_radius_m)
    |   movel([0.154089, -0.767013, -2.807856, -1.137520, 1.570796, 1.724885],accel_mss,speed_ms,0,blend_radius_m)
    |   movel([0.159674, -0.769070, -2.807547, -1.135772, 1.570796, 1.730470],accel_mss,speed_ms,0,blend_radius_m)
    |   movel([0.162746, -0.770389, -2.807348, -1.134652, 1.570796, 1.733543],accel_mss,speed_ms,0,blend_radius_m)
    |   movel([0.163612, -0.771116, -2.807239, -1.134035, 1.570796, 1.734409],accel_mss,speed_ms,0,blend_radius_m)
    |   movel([0.163756, -0.771883, -2.807122, -1.133384, 1.570796, 1.734553],accel_mss,speed_ms,0,blend_radius_m)
    |   movel([0.163286, -0.772807, -2.806982, -1.132600, 1.570796, 1.734082],accel_mss,speed_ms,0,blend_radius_m)
    |   movel([0.162613, -0.773696, -2.806846, -1.131846, 1.570796, 1.733409],accel_mss,speed_ms,0,blend_radius_m)
    |   movel([0.161019, -0.775085, -2.806634, -1.130670, 1.570796, 1.731815],accel_mss,speed_ms,0,blend_radius_m)
    |   movel([0.159729, -0.775716, -2.806537, -1.130136, 1.570796, 1.730525],accel_mss,speed_ms,0,blend_radius_m)
    |   movel([0.158459, -0.776086, -2.806480, -1.129823, 1.570796, 1.729255],accel_mss,speed_ms,0,blend_radius_m)
    |   movel([0.156067, -0.776580, -2.806404, -1.129405, 1.570796, 1.726863],accel_mss,speed_ms,0,blend_radius_m)
    |   movel([0.156904, -0.779688, -2.805923, -1.126779, 1.570796, 1.727700],accel_mss,speed_ms,0,blend_radius_m)
    |   movel([0.158028, -0.782503, -2.805483, -1.124404, 1.570796, 1.728824],accel_mss,speed_ms,0,blend_radius_m)
    |   movel([0.159435, -0.785013, -2.805087, -1.122289, 1.570796, 1.730231],accel_mss,speed_ms,0,blend_radius_m)
    |   movel([0.161100, -0.787223, -2.804736, -1.120430, 1.570796, 1.731897],accel_mss,speed_ms,0,blend_radius_m)
    |   movel([0.163153, -0.788903, -2.804467, -1.119019, 1.570796, 1.733950],accel_mss,speed_ms,0,blend_radius_m)
    |   movel([0.165632, -0.790001, -2.804291, -1.118097, 1.570796, 1.736429],accel_mss,speed_ms,0,blend_radius_m)
    |   movel([0.171148, -0.791356, -2.804073, -1.116960, 1.570796, 1.741945],accel_mss,speed_ms,0,blend_radius_m)
    |   movel([0.172518, -0.792096, -2.803953, -1.116340, 1.570796, 1.743314],accel_mss,speed_ms,0,blend_radius_m)
    |   movel([0.172777, -0.792875, -2.803827, -1.115687, 1.570796, 1.743574],accel_mss,speed_ms,0,blend_radius_m)
    |   movel([0.172510, -0.794022, -2.803640, -1.114726, 1.570796, 1.743306],accel_mss,speed_ms,0,blend_radius_m)
    |   movel([0.171843, -0.795144, -2.803457, -1.113788, 1.570796, 1.742640],accel_mss,speed_ms,0,blend_radius_m)
    |   movel([0.170946, -0.796146, -2.803293, -1.112949, 1.570796, 1.741743],accel_mss,speed_ms,0,blend_radius_m)
    |   movel([0.168898, -0.797743, -2.803031, -1.111615, 1.570796, 1.739694],accel_mss,speed_ms,0,blend_radius_m)
    |   movel([0.166230, -0.799302, -2.802774, -1.110314, 1.570796, 1.737027],accel_mss,speed_ms,0,blend_radius_m)
    |   movel([0.163684, -0.800483, -2.802578, -1.109328, 1.570796, 1.734480],accel_mss,speed_ms,0,blend_radius_m)
    |   movel([0.161241, -0.801346, -2.802434, -1.108609, 1.570796, 1.732037],accel_mss,speed_ms,0,blend_radius_m)
    |   movel([0.158895, -0.801926, -2.802338, -1.108125, 1.570796, 1.729691],accel_mss,speed_ms,0,blend_radius_m)
    |   movel([0.160207, -0.804042, -2.801983, -1.106364, 1.570796, 1.731003],accel_mss,speed_ms,0,blend_radius_m)
    |   movel([0.161845, -0.805747, -2.801696, -1.104946, 1.570796, 1.732641],accel_mss,speed_ms,0,blend_radius_m)
    |   movel([0.163803, -0.806996, -2.801485, -1.103908, 1.570796, 1.734600],accel_mss,speed_ms,0,blend_radius_m)
    |   movel([0.166076, -0.807752, -2.801357, -1.103280, 1.570796, 1.736872],accel_mss,speed_ms,0,blend_radius_m)
    |   movel([0.168667, -0.807965, -2.801320, -1.103103, 1.570796, 1.739463],accel_mss,speed_ms,0,blend_radius_m)
    |   movel([0.171579, -0.807593, -2.801384, -1.103412, 1.570796, 1.742375],accel_mss,speed_ms,0,blend_radius_m)
    |   movel([0.174810, -0.806585, -2.801555, -1.104250, 1.570796, 1.745606],accel_mss,speed_ms,0,blend_radius_m)
    |   movel([0.178370, -0.804894, -2.801840, -1.105655, 1.570796, 1.749166],accel_mss,speed_ms,0,blend_radius_m)
    |   speed_ms = 0.005
    |   movel([0.178370, -0.796314, -2.795475, -1.120600, 1.570796, 1.749166],accel_mss,speed_ms,0,blend_radius_m)
    |   speed_ms = 0.040
    |   movel([0.194494, -0.771439, -2.799476, -1.141474, 1.570796, 1.765291],accel_mss,speed_ms,0,blend_radius_m)
    |   speed_ms = 0.005
    |   movel([0.194494, -0.779746, -2.805914, -1.126730, 1.570796, 1.765291],accel_mss,speed_ms,0,blend_radius_m)
    |   speed_ms = 0.025
    |   movel([0.187997, -0.779767, -2.805910, -1.126711, 1.570796, 1.758793],accel_mss,speed_ms,0,blend_radius_m)
    |   movel([0.185246, -0.779451, -2.805959, -1.126978, 1.570796, 1.756042],accel_mss,speed_ms,0,blend_radius_m)
    |   movel([0.182809, -0.778809, -2.806059, -1.127521, 1.570796, 1.753606],accel_mss,speed_ms,0,blend_radius_m)
    |   movel([0.180667, -0.777755, -2.806223, -1.128412, 1.570796, 1.751463],accel_mss,speed_ms,0,blend_radius_m)
    |   movel([0.178806, -0.776207, -2.806461, -1.129721, 1.570796, 1.749602],accel_mss,speed_ms,0,blend_radius_m)
    |   movel([0.177203, -0.774090, -2.806786, -1.131513, 1.570796, 1.748000],accel_mss,speed_ms,0,blend_radius_m)
    |   movel([0.175851, -0.771313, -2.807209, -1.133867, 1.570796, 1.746648],accel_mss,speed_ms,0,blend_radius_m)
    |   movel([0.173805, -0.764717, -2.808197, -1.139475, 1.570796, 1.744601],accel_mss,speed_ms,0,blend_radius_m)
    |   movel([0.172497, -0.757377, -2.809273, -1.145739, 1.570796, 1.743293],accel_mss,speed_ms,0,blend_radius_m)
    |   movel([0.171862, -0.749383, -2.810415, -1.152591, 1.570796, 1.742658],accel_mss,speed_ms,0,blend_radius_m)
    |   movel([0.171826, -0.740848, -2.811601, -1.159940, 1.570796, 1.742622],accel_mss,speed_ms,0,blend_radius_m)
    |   movel([0.172236, -0.733482, -2.812598, -1.166309, 1.570796, 1.743032],accel_mss,speed_ms,0,blend_radius_m)
    |   movel([0.173002, -0.725814, -2.813609, -1.172966, 1.570796, 1.743798],accel_mss,speed_ms,0,blend_radius_m)
    |   movel([0.175347, -0.709737, -2.815642, -1.187010, 1.570796, 1.746143],accel_mss,speed_ms,0,blend_radius_m)
    |   movel([0.185575, -0.651688, -2.822049, -1.238651, 1.570796, 1.756371],accel_mss,speed_ms,0,blend_radius_m)
    |   movel([0.187754, -0.639201, -2.823244, -1.249944, 1.570796, 1.758551],accel_mss,speed_ms,0,blend_radius_m)
    |   movel([0.189739, -0.626743, -2.824374, -1.261272, 1.570796, 1.760536],accel_mss,speed_ms,0,blend_radius_m)
    |   movel([0.191349, -0.614506, -2.825425, -1.272458, 1.570796, 1.762145],accel_mss,speed_ms,0,blend_radius_m)
    |   movel([0.192388, -0.602675, -2.826385, -1.283329, 1.570796, 1.763185],accel_mss,speed_ms,0,blend_radius_m)
    |   movel([0.192664, -0.591456, -2.827246, -1.293687, 1.570796, 1.763460],accel_mss,speed_ms,0,blend_radius_m)
    |   movel([0.191964, -0.581069, -2.828000, -1.303320, 1.570796, 1.762760],accel_mss,speed_ms,0,blend_radius_m)
    |   movel([0.190761, -0.574126, -2.828482, -1.309781, 1.570796, 1.761557],accel_mss,speed_ms,0,blend_radius_m)
    |   movel([0.188920, -0.567574, -2.828921, -1.315894, 1.570796, 1.759717],accel_mss,speed_ms,0,blend_radius_m)
    |   movel([0.186387, -0.561607, -2.829306, -1.321476, 1.570796, 1.757184],accel_mss,speed_ms,0,blend_radius_m)
    |   movel([0.183102, -0.556416, -2.829631, -1.326342, 1.570796, 1.753899],accel_mss,speed_ms,0,blend_radius_m)
    |   movel([0.179022, -0.552184, -2.829888, -1.330316, 1.570796, 1.749818],accel_mss,speed_ms,0,blend_radius_m)
    |   movel([0.174102, -0.549091, -2.830072, -1.333225, 1.570796, 1.744898],accel_mss,speed_ms,0,blend_radius_m)
    |   movel([0.168297, -0.547333, -2.830176, -1.334880, 1.570796, 1.739093],accel_mss,speed_ms,0,blend_radius_m)
    |   movel([0.161591, -0.547073, -2.830191, -1.335126, 1.570796, 1.732387],accel_mss,speed_ms,0,blend_radius_m)
    |   movel([0.158088, -0.547578, -2.830161, -1.334650, 1.570796, 1.728885],accel_mss,speed_ms,0,blend_radius_m)
    |   movel([0.154299, -0.548579, -2.830103, -1.333707, 1.570796, 1.725095],accel_mss,speed_ms,0,blend_radius_m)
    |   movel([0.150252, -0.550098, -2.830013, -1.332278, 1.570796, 1.721048],accel_mss,speed_ms,0,blend_radius_m)
    |   movel([0.145990, -0.552141, -2.829891, -1.330357, 1.570796, 1.716787],accel_mss,speed_ms,0,blend_radius_m)
    |   movel([0.141561, -0.554705, -2.829736, -1.327949, 1.570796, 1.712357],accel_mss,speed_ms,0,blend_radius_m)
    |   movel([0.136989, -0.557814, -2.829544, -1.325030, 1.570796, 1.707786],accel_mss,speed_ms,0,blend_radius_m)
    |   movel([0.132330, -0.561456, -2.829316, -1.321617, 1.570796, 1.703126],accel_mss,speed_ms,0,blend_radius_m)
    |   movel([0.127623, -0.565643, -2.829047, -1.317699, 1.570796, 1.698420],accel_mss,speed_ms,0,blend_radius_m)
    |   speed_ms = 0.005
    |   movel([0.127623, -0.560504, -2.822160, -1.329725, 1.570796, 1.698420],accel_mss,speed_ms,0,blend_radius_m)
    |   speed_ms = 0.040
    |   movel([0.112521, -0.547930, -2.822945, -1.341514, 1.570796, 1.683317],accel_mss,speed_ms,0,blend_radius_m)
    |   speed_ms = 0.005
    |   movel([0.112521, -0.552838, -2.829849, -1.329702, 1.570796, 1.683317],accel_mss,speed_ms,0,blend_radius_m)
    |   speed_ms = 0.025
    |   movel([0.112052, -0.550367, -2.829997, -1.332025, 1.570796, 1.682848],accel_mss,speed_ms,0,blend_radius_m)
    |   movel([0.111963, -0.547554, -2.830163, -1.334673, 1.570796, 1.682759],accel_mss,speed_ms,0,blend_radius_m)
    |   movel([0.112709, -0.541121, -2.830531, -1.340737, 1.570796, 1.683505],accel_mss,speed_ms,0,blend_radius_m)
    |   movel([0.114351, -0.533929, -2.830925, -1.347534, 1.570796, 1.685147],accel_mss,speed_ms,0,blend_radius_m)
    |   movel([0.116452, -0.526409, -2.831318, -1.354662, 1.570796, 1.687249],accel_mss,speed_ms,0,blend_radius_m)
    |   speed_ms = 0.005
    |   movel([0.116452, -0.521990, -2.824383, -1.366017, 1.570796, 1.687249],accel_mss,speed_ms,0,blend_radius_m)
    |   speed_ms = 0.040
    |   movel([0.126566, -0.517944, -2.824585, -1.369860, 1.570796, 1.697362],accel_mss,speed_ms,0,blend_radius_m)
    |   speed_ms = 0.005
    |   movel([0.126566, -0.522286, -2.831524, -1.358578, 1.570796, 1.697362],accel_mss,speed_ms,0,blend_radius_m)
    |   speed_ms = 0.025
    |   movel([0.125324, -0.520855, -2.831595, -1.359939, 1.570796, 1.696121],accel_mss,speed_ms,0,blend_radius_m)
    |   movel([0.124468, -0.519068, -2.831681, -1.361639, 1.570796, 1.695264],accel_mss,speed_ms,0,blend_radius_m)
    |   movel([0.123806, -0.514519, -2.831897, -1.365973, 1.570796, 1.694602],accel_mss,speed_ms,0,blend_radius_m)
    |   movel([0.124407, -0.508847, -2.832156, -1.371385, 1.570796, 1.695203],accel_mss,speed_ms,0,blend_radius_m)
    |   movel([0.126097, -0.502249, -2.832444, -1.377696, 1.570796, 1.696894],accel_mss,speed_ms,0,blend_radius_m)
    |   movel([0.128698, -0.494936, -2.832744, -1.384709, 1.570796, 1.699495],accel_mss,speed_ms,0,blend_radius_m)
    |   movel([0.132025, -0.487127, -2.833045, -1.392217, 1.570796, 1.702822],accel_mss,speed_ms,0,blend_radius_m)
    |   movel([0.135889, -0.479044, -2.833335, -1.400010, 1.570796, 1.706685],accel_mss,speed_ms,0,blend_radius_m)
    |   movel([0.140087, -0.470924, -2.833603, -1.407862, 1.570796, 1.710884],accel_mss,speed_ms,0,blend_radius_m)
    |   speed_ms = 0.005
    |   movel([0.140087, -0.467577, -2.826620, -1.418193, 1.570796, 1.710884],accel_mss,speed_ms,0,blend_radius_m)
    |   speed_ms = 0.040
    |   movel([0.195766, -0.390545, -2.828046, -1.493798, 1.570796, 1.766562],accel_mss,speed_ms,0,blend_radius_m)
    |   speed_ms = 0.005
    |   movel([0.195766, -0.392285, -2.835060, -1.485044, 1.570796, 1.766562],accel_mss,speed_ms,0,blend_radius_m)
    |   speed_ms = 0.025
    |   movel([0.190041, -0.398855, -2.835017, -1.478517, 1.570796, 1.760837],accel_mss,speed_ms,0,blend_radius_m)
    |   movel([0.184352, -0.405749, -2.834956, -1.471684, 1.570796, 1.755149],accel_mss,speed_ms,0,blend_radius_m)
    |   movel([0.178795, -0.412855, -2.834877, -1.464658, 1.570796, 1.749591],accel_mss,speed_ms,0,blend_radius_m)
    |   movel([0.173431, -0.420090, -2.834779, -1.457520, 1.570796, 1.744228],accel_mss,speed_ms,0,blend_radius_m)
    |   movel([0.168353, -0.427356, -2.834664, -1.450369, 1.570796, 1.739150],accel_mss,speed_ms,0,blend_radius_m)
    |   movel([0.163627, -0.434558, -2.834532, -1.443299, 1.570796, 1.734423],accel_mss,speed_ms,0,blend_radius_m)
    |   movel([0.159325, -0.441617, -2.834386, -1.436386, 1.570796, 1.730121],accel_mss,speed_ms,0,blend_radius_m)
    |   movel([0.155512, -0.448450, -2.834229, -1.429709, 1.570796, 1.726308],accel_mss,speed_ms,0,blend_radius_m)
    |   movel([0.152251, -0.454966, -2.834065, -1.423358, 1.570796, 1.723047],accel_mss,speed_ms,0,blend_radius_m)
    |   movel([0.149600, -0.461099, -2.833898, -1.417392, 1.570796, 1.720396],accel_mss,speed_ms,0,blend_radius_m)
    |   movel([0.147616, -0.466770, -2.833732, -1.411888, 1.570796, 1.718412],accel_mss,speed_ms,0,blend_radius_m)
    |   movel([0.146355, -0.471906, -2.833572, -1.406911, 1.570796, 1.717152],accel_mss,speed_ms,0,blend_radius_m)
    |   movel([0.145880, -0.476431, -2.833423, -1.402534, 1.570796, 1.716676],accel_mss,speed_ms,0,blend_radius_m)
    |   movel([0.146245, -0.480277, -2.833292, -1.398820, 1.570796, 1.717041],accel_mss,speed_ms,0,blend_radius_m)
    |   movel([0.147498, -0.483382, -2.833182, -1.395825, 1.570796, 1.718294],accel_mss,speed_ms,0,blend_radius_m)
    |   movel([0.149705, -0.485672, -2.833099, -1.393618, 1.570796, 1.720501],accel_mss,speed_ms,0,blend_radius_m)
    |   speed_ms = 0.005
    |   movel([0.149705, -0.482034, -2.826126, -1.404229, 1.570796, 1.720501],accel_mss,speed_ms,0,blend_radius_m)
    |   speed_ms = 0.040
    |   movel([0.174765, -0.454061, -2.827015, -1.431312, 1.570796, 1.745561],accel_mss,speed_ms,0,blend_radius_m)
    |   speed_ms = 0.005
    |   movel([0.174765, -0.457133, -2.834007, -1.421248, 1.570796, 1.745561],accel_mss,speed_ms,0,blend_radius_m)
    |   speed_ms = 0.025
    |   movel([0.174309, -0.454103, -2.834088, -1.424198, 1.570796, 1.745105],accel_mss,speed_ms,0,blend_radius_m)
    |   movel([0.174262, -0.450672, -2.834175, -1.427542, 1.570796, 1.745059],accel_mss,speed_ms,0,blend_radius_m)
    |   movel([0.174623, -0.446879, -2.834267, -1.431244, 1.570796, 1.745419],accel_mss,speed_ms,0,blend_radius_m)
    |   movel([0.175391, -0.442742, -2.834361, -1.435285, 1.570796, 1.746187],accel_mss,speed_ms,0,blend_radius_m)
    |   movel([0.176558, -0.438301, -2.834457, -1.439631, 1.570796, 1.747354],accel_mss,speed_ms,0,blend_radius_m)
    |   movel([0.178133, -0.433576, -2.834551, -1.444262, 1.570796, 1.748929],accel_mss,speed_ms,0,blend_radius_m)
    |   movel([0.180117, -0.428586, -2.834642, -1.449161, 1.570796, 1.750913],accel_mss,speed_ms,0,blend_radius_m)
    |   movel([0.182501, -0.423378, -2.834729, -1.454282, 1.570796, 1.753297],accel_mss,speed_ms,0,blend_radius_m)
    |   movel([0.185287, -0.417973, -2.834809, -1.459606, 1.570796, 1.756083],accel_mss,speed_ms,0,blend_radius_m)
    |   movel([0.188481, -0.412394, -2.834882, -1.465113, 1.570796, 1.759278],accel_mss,speed_ms,0,blend_radius_m)
    |   movel([0.192066, -0.406695, -2.834946, -1.470748, 1.570796, 1.762862],accel_mss,speed_ms,0,blend_radius_m)
    |   movel([0.196058, -0.400881, -2.835000, -1.476507, 1.570796, 1.766854],accel_mss,speed_ms,0,blend_radius_m)
    |   movel([0.200445, -0.394998, -2.835044, -1.482347, 1.570796, 1.771241],accel_mss,speed_ms,0,blend_radius_m)
    |   movel([0.205224, -0.389078, -2.835077, -1.488234, 1.570796, 1.776020],accel_mss,speed_ms,0,blend_radius_m)
    |   movel([0.210387, -0.383164, -2.835098, -1.494127, 1.570796, 1.781183],accel_mss,speed_ms,0,blend_radius_m)
    |   movel([0.215921, -0.377293, -2.835107, -1.499989, 1.570796, 1.786717],accel_mss,speed_ms,0,blend_radius_m)
    |   movel([0.221470, -0.371861, -2.835106, -1.505421, 1.570796, 1.792267],accel_mss,speed_ms,0,blend_radius_m)
    |   movel([0.226986, -0.366900, -2.835097, -1.510392, 1.570796, 1.797782],accel_mss,speed_ms,0,blend_radius_m)
    |   movel([0.232424, -0.362417, -2.835081, -1.514891, 1.570796, 1.803221],accel_mss,speed_ms,0,blend_radius_m)
    |   movel([0.237763, -0.358415, -2.835062, -1.518912, 1.570796, 1.808559],accel_mss,speed_ms,0,blend_radius_m)
    |   movel([0.242958, -0.354900, -2.835041, -1.522447, 1.570796, 1.813755],accel_mss,speed_ms,0,blend_radius_m)
    |   movel([0.247964, -0.351894, -2.835020, -1.525475, 1.570796, 1.818760],accel_mss,speed_ms,0,blend_radius_m)
    |   movel([0.252766, -0.349373, -2.835000, -1.528016, 1.570796, 1.823562],accel_mss,speed_ms,0,blend_radius_m)
    |   movel([0.257302, -0.347368, -2.834982, -1.530038, 1.570796, 1.828098],accel_mss,speed_ms,0,blend_radius_m)
    |   movel([0.261557, -0.345869, -2.834969, -1.531551, 1.570796, 1.832353],accel_mss,speed_ms,0,blend_radius_m)
    |   movel([0.269094, -0.344375, -2.834954, -1.533060, 1.570796, 1.839891],accel_mss,speed_ms,0,blend_radius_m)
    |   movel([0.272303, -0.344389, -2.834954, -1.533046, 1.570796, 1.843099],accel_mss,speed_ms,0,blend_radius_m)
    |   movel([0.277502, -0.345887, -2.834969, -1.531533, 1.570796, 1.848299],accel_mss,speed_ms,0,blend_radius_m)
    |   movel([0.279440, -0.347357, -2.834982, -1.530049, 1.570796, 1.850237],accel_mss,speed_ms,0,blend_radius_m)
    |   movel([0.280900, -0.349303, -2.834999, -1.528086, 1.570796, 1.851696],accel_mss,speed_ms,0,blend_radius_m)
    |   speed_ms = 0.005
    |   movel([0.280900, -0.348474, -2.827986, -1.535930, 1.570796, 1.851696],accel_mss,speed_ms,0,blend_radius_m)
    |   speed_ms = 0.040
    |   movel([0.297437, -0.361211, -2.828066, -1.523112, 1.570796, 1.868234],accel_mss,speed_ms,0,blend_radius_m)
    |   speed_ms = 0.005
    |   movel([0.297437, -0.362318, -2.835081, -1.514990, 1.570796, 1.868234],accel_mss,speed_ms,0,blend_radius_m)
    |   speed_ms = 0.025
    |   movel([0.295487, -0.359060, -2.835066, -1.518264, 1.570796, 1.866283],accel_mss,speed_ms,0,blend_radius_m)
    |   movel([0.292449, -0.357093, -2.835055, -1.520241, 1.570796, 1.863246],accel_mss,speed_ms,0,blend_radius_m)
    |   movel([0.288405, -0.356411, -2.835051, -1.520928, 1.570796, 1.859202],accel_mss,speed_ms,0,blend_radius_m)
    |   movel([0.283424, -0.357006, -2.835054, -1.520329, 1.570796, 1.854220],accel_mss,speed_ms,0,blend_radius_m)
    |   movel([0.277622, -0.358841, -2.835065, -1.518483, 1.570796, 1.848419],accel_mss,speed_ms,0,blend_radius_m)
    |   movel([0.271084, -0.361904, -2.835079, -1.515406, 1.570796, 1.841880],accel_mss,speed_ms,0,blend_radius_m)
    |   movel([0.263932, -0.366146, -2.835095, -1.511148, 1.570796, 1.834728],accel_mss,speed_ms,0,blend_radius_m)
    |   movel([0.256265, -0.371534, -2.835106, -1.505749, 1.570796, 1.827061],accel_mss,speed_ms,0,blend_radius_m)
    |   movel([0.248224, -0.378004, -2.835107, -1.499278, 1.570796, 1.819020],accel_mss,speed_ms,0,blend_radius_m)
    |   movel([0.240005, -0.385423, -2.835091, -1.491875, 1.570796, 1.810802],accel_mss,speed_ms,0,blend_radius_m)
    |   movel([0.231940, -0.393517, -2.835053, -1.483819, 1.570796, 1.802736],accel_mss,speed_ms,0,blend_radius_m)
    |   movel([0.224362, -0.402021, -2.834991, -1.475377, 1.570796, 1.795158],accel_mss,speed_ms,0,blend_radius_m)
    |   movel([0.217560, -0.410699, -2.834902, -1.466787, 1.570796, 1.788356],accel_mss,speed_ms,0,blend_radius_m)
    |   movel([0.214549, -0.415021, -2.834849, -1.462519, 1.570796, 1.785346],accel_mss,speed_ms,0,blend_radius_m)
    |   movel([0.211837, -0.419295, -2.834791, -1.458304, 1.570796, 1.782633],accel_mss,speed_ms,0,blend_radius_m)
    |   movel([0.209456, -0.423497, -2.834727, -1.454164, 1.570796, 1.780253],accel_mss,speed_ms,0,blend_radius_m)
    |   movel([0.207448, -0.427603, -2.834659, -1.450127, 1.570796, 1.778244],accel_mss,speed_ms,0,blend_radius_m)
    |   movel([0.205832, -0.431582, -2.834588, -1.446219, 1.570796, 1.776628],accel_mss,speed_ms,0,blend_radius_m)
    |   movel([0.204656, -0.435397, -2.834515, -1.442477, 1.570796, 1.775453],accel_mss,speed_ms,0,blend_radius_m)
    |   speed_ms = 0.005
    |   movel([0.204656, -0.432765, -2.827513, -1.452112, 1.570796, 1.775453],accel_mss,speed_ms,0,blend_radius_m)
    |   speed_ms = 0.040
    |   movel([0.242771, -0.419080, -2.827751, -1.465558, 1.570796, 1.813567],accel_mss,speed_ms,0,blend_radius_m)
    |   speed_ms = 0.005
    |   movel([0.242771, -0.421426, -2.834759, -1.456204, 1.570796, 1.813567],accel_mss,speed_ms,0,blend_radius_m)
    |   speed_ms = 0.025
    |   movel([0.248268, -0.415291, -2.834846, -1.462253, 1.570796, 1.819065],accel_mss,speed_ms,0,blend_radius_m)
    |   movel([0.253942, -0.409638, -2.834915, -1.467836, 1.570796, 1.824739],accel_mss,speed_ms,0,blend_radius_m)
    |   movel([0.259702, -0.404503, -2.834968, -1.472919, 1.570796, 1.830499],accel_mss,speed_ms,0,blend_radius_m)
    |   movel([0.265431, -0.399943, -2.835008, -1.477438, 1.570796, 1.836228],accel_mss,speed_ms,0,blend_radius_m)
    |   movel([0.271029, -0.396000, -2.835037, -1.481352, 1.570796, 1.841825],accel_mss,speed_ms,0,blend_radius_m)
    |   movel([0.276380, -0.392716, -2.835058, -1.484615, 1.570796, 1.847177],accel_mss,speed_ms,0,blend_radius_m)
    |   movel([0.281392, -0.390128, -2.835072, -1.487189, 1.570796, 1.852188],accel_mss,speed_ms,0,blend_radius_m)
    |   movel([0.285943, -0.388281, -2.835080, -1.489028, 1.570796, 1.856740],accel_mss,speed_ms,0,blend_radius_m)
    |   movel([0.290676, -0.387225, -2.835084, -1.490080, 1.570796, 1.861472],accel_mss,speed_ms,0,blend_radius_m)
    |   movel([0.294007, -0.387680, -2.835083, -1.489627, 1.570796, 1.864803],accel_mss,speed_ms,0,blend_radius_m)
    |   movel([0.296088, -0.389479, -2.835075, -1.487836, 1.570796, 1.866884],accel_mss,speed_ms,0,blend_radius_m)
    |   movel([0.297048, -0.392475, -2.835059, -1.484855, 1.570796, 1.867844],accel_mss,speed_ms,0,blend_radius_m)
    |   movel([0.297043, -0.396485, -2.835034, -1.480870, 1.570796, 1.867839],accel_mss,speed_ms,0,blend_radius_m)
    |   movel([0.296222, -0.401356, -2.834996, -1.476036, 1.570796, 1.867018],accel_mss,speed_ms,0,blend_radius_m)
    |   movel([0.294732, -0.406920, -2.834944, -1.470525, 1.570796, 1.865528],accel_mss,speed_ms,0,blend_radius_m)
    |   movel([0.292732, -0.413007, -2.834875, -1.464507, 1.570796, 1.863528],accel_mss,speed_ms,0,blend_radius_m)
    |   speed_ms = 0.005
    |   movel([0.292732, -0.410835, -2.827864, -1.473690, 1.570796, 1.863528],accel_mss,speed_ms,0,blend_radius_m)
    |   speed_ms = 0.040
    |   movel([0.255676, -0.434165, -2.827485, -1.450739, 1.570796, 1.826472],accel_mss,speed_ms,0,blend_radius_m)
    |   speed_ms = 0.005
    |   movel([0.255676, -0.436826, -2.834487, -1.441076, 1.570796, 1.826472],accel_mss,speed_ms,0,blend_radius_m)
    |   speed_ms = 0.025
    |   movel([0.260590, -0.434034, -2.834542, -1.443813, 1.570796, 1.831386],accel_mss,speed_ms,0,blend_radius_m)
    |   movel([0.265016, -0.432025, -2.834580, -1.445784, 1.570796, 1.835812],accel_mss,speed_ms,0,blend_radius_m)
    |   movel([0.268950, -0.430782, -2.834603, -1.447003, 1.570796, 1.839746],accel_mss,speed_ms,0,blend_radius_m)
    |   movel([0.272400, -0.430254, -2.834613, -1.447522, 1.570796, 1.843197],accel_mss,speed_ms,0,blend_radius_m)
    |   movel([0.275371, -0.430413, -2.834610, -1.447367, 1.570796, 1.846167],accel_mss,speed_ms,0,blend_radius_m)
    |   movel([0.277866, -0.431213, -2.834595, -1.446581, 1.570796, 1.848663],accel_mss,speed_ms,0,blend_radius_m)
    |   movel([0.279904, -0.432612, -2.834569, -1.445208, 1.570796, 1.850701],accel_mss,speed_ms,0,blend_radius_m)
    |   movel([0.281481, -0.434582, -2.834531, -1.443276, 1.570796, 1.852278],accel_mss,speed_ms,0,blend_radius_m)
    |   movel([0.282628, -0.437063, -2.834482, -1.440844, 1.570796, 1.853425],accel_mss,speed_ms,0,blend_radius_m)
    |   movel([0.283355, -0.440013, -2.834421, -1.437955, 1.570796, 1.854151],accel_mss,speed_ms,0,blend_radius_m)
    |   movel([0.283668, -0.443396, -2.834347, -1.434646, 1.570796, 1.854465],accel_mss,speed_ms,0,blend_radius_m)
    |   movel([0.283595, -0.447157, -2.834260, -1.430971, 1.570796, 1.854391],accel_mss,speed_ms,0,blend_radius_m)
    |   movel([0.283144, -0.451260, -2.834160, -1.426969, 1.570796, 1.853941],accel_mss,speed_ms,0,blend_radius_m)
    |   movel([0.281185, -0.460295, -2.833920, -1.418174, 1.570796, 1.851982],accel_mss,speed_ms,0,blend_radius_m)
    |   movel([0.279703, -0.465150, -2.833780, -1.413459, 1.570796, 1.850500],accel_mss,speed_ms,0,blend_radius_m)
    |   movel([0.279603, -0.463954, -2.833815, -1.414620, 1.570796, 1.850399],accel_mss,speed_ms,0,blend_radius_m)
    |   speed_ms = 0.005
    |   movel([0.279603, -0.460745, -2.826828, -1.424816, 1.570796, 1.850399],accel_mss,speed_ms,0,blend_radius_m)
    |   speed_ms = 0.040
    |   movel([0.306953, -0.457953, -2.826908, -1.427528, 1.570796, 1.877749],accel_mss,speed_ms,0,blend_radius_m)
    |   speed_ms = 0.005
    |   movel([0.306953, -0.461104, -2.833898, -1.417387, 1.570796, 1.877749],accel_mss,speed_ms,0,blend_radius_m)
    |   speed_ms = 0.025
    |   movel([0.301707, -0.469174, -2.833658, -1.409557, 1.570796, 1.872503],accel_mss,speed_ms,0,blend_radius_m)
    |   movel([0.297075, -0.477100, -2.833401, -1.401888, 1.570796, 1.867872],accel_mss,speed_ms,0,blend_radius_m)
    |   movel([0.292933, -0.484866, -2.833128, -1.394395, 1.570796, 1.863729],accel_mss,speed_ms,0,blend_radius_m)
    |   movel([0.289143, -0.492465, -2.832842, -1.387082, 1.570796, 1.859939],accel_mss,speed_ms,0,blend_radius_m)
    |   movel([0.285336, -0.500645, -2.832511, -1.379233, 1.570796, 1.856132],accel_mss,speed_ms,0,blend_radius_m)
    |   movel([0.283763, -0.504542, -2.832346, -1.375501, 1.570796, 1.854559],accel_mss,speed_ms,0,blend_radius_m)
    |   movel([0.282543, -0.508221, -2.832184, -1.371984, 1.570796, 1.853339],accel_mss,speed_ms,0,blend_radius_m)
    |   movel([0.281764, -0.511606, -2.832032, -1.368752, 1.570796, 1.852560],accel_mss,speed_ms,0,blend_radius_m)
    |   movel([0.281531, -0.514547, -2.831896, -1.365946, 1.570796, 1.852327],accel_mss,speed_ms,0,blend_radius_m)
    |   movel([0.281942, -0.516855, -2.831787, -1.363747, 1.570796, 1.852738],accel_mss,speed_ms,0,blend_radius_m)
    |   movel([0.283072, -0.518378, -2.831715, -1.362297, 1.570796, 1.853869],accel_mss,speed_ms,0,blend_radius_m)
    |   movel([0.285994, -0.519338, -2.831668, -1.361383, 1.570796, 1.856791],accel_mss,speed_ms,0,blend_radius_m)
    |   movel([0.287429, -0.519839, -2.831644, -1.360906, 1.570796, 1.858226],accel_mss,speed_ms,0,blend_radius_m)
    |   movel([0.288478, -0.520820, -2.831596, -1.359973, 1.570796, 1.859275],accel_mss,speed_ms,0,blend_radius_m)
    |   movel([0.288875, -0.522885, -2.831495, -1.358009, 1.570796, 1.859671],accel_mss,speed_ms,0,blend_radius_m)
    |   movel([0.288483, -0.525894, -2.831344, -1.355152, 1.570796, 1.859279],accel_mss,speed_ms,0,blend_radius_m)
    |   movel([0.287486, -0.529592, -2.831154, -1.351643, 1.570796, 1.858282],accel_mss,speed_ms,0,blend_radius_m)
    |   movel([0.286055, -0.533725, -2.830936, -1.347728, 1.570796, 1.856851],accel_mss,speed_ms,0,blend_radius_m)
    |   movel([0.282563, -0.542323, -2.830463, -1.339602, 1.570796, 1.853360],accel_mss,speed_ms,0,blend_radius_m)
    |   movel([0.271861, -0.566484, -2.828992, -1.316913, 1.570796, 1.842658],accel_mss,speed_ms,0,blend_radius_m)
    |   movel([0.264682, -0.582902, -2.827870, -1.301617, 1.570796, 1.835478],accel_mss,speed_ms,0,blend_radius_m)
    |   movel([0.262800, -0.587778, -2.827518, -1.297094, 1.570796, 1.833596],accel_mss,speed_ms,0,blend_radius_m)
    |   movel([0.261094, -0.592833, -2.827143, -1.292414, 1.570796, 1.831890],accel_mss,speed_ms,0,blend_radius_m)
    |   movel([0.258380, -0.603034, -2.826356, -1.282999, 1.570796, 1.829176],accel_mss,speed_ms,0,blend_radius_m)
    |   movel([0.257462, -0.607958, -2.825963, -1.278468, 1.570796, 1.828258],accel_mss,speed_ms,0,blend_radius_m)
    |   movel([0.256893, -0.612617, -2.825581, -1.274190, 1.570796, 1.827690],accel_mss,speed_ms,0,blend_radius_m)
    |   movel([0.256711, -0.616907, -2.825223, -1.270259, 1.570796, 1.827508],accel_mss,speed_ms,0,blend_radius_m)
    |   movel([0.256956, -0.620728, -2.824898, -1.266763, 1.570796, 1.827752],accel_mss,speed_ms,0,blend_radius_m)
    |   movel([0.257672, -0.623962, -2.824618, -1.263809, 1.570796, 1.828468],accel_mss,speed_ms,0,blend_radius_m)
    |   movel([0.258891, -0.626526, -2.824393, -1.261470, 1.570796, 1.829687],accel_mss,speed_ms,0,blend_radius_m)
    |   movel([0.260666, -0.628299, -2.824236, -1.259854, 1.570796, 1.831462],accel_mss,speed_ms,0,blend_radius_m)
    |   movel([0.263036, -0.629183, -2.824158, -1.259048, 1.570796, 1.833832],accel_mss,speed_ms,0,blend_radius_m)
    |   movel([0.266044, -0.629074, -2.824168, -1.259148, 1.570796, 1.836840],accel_mss,speed_ms,0,blend_radius_m)
    |   movel([0.269749, -0.627854, -2.824276, -1.260259, 1.570796, 1.840545],accel_mss,speed_ms,0,blend_radius_m)
    |   movel([0.274203, -0.625414, -2.824491, -1.262484, 1.570796, 1.844999],accel_mss,speed_ms,0,blend_radius_m)
    |   movel([0.279471, -0.621632, -2.824820, -1.265937, 1.570796, 1.850267],accel_mss,speed_ms,0,blend_radius_m)
    |   movel([0.283689, -0.618071, -2.825125, -1.269193, 1.570796, 1.854485],accel_mss,speed_ms,0,blend_radius_m)
    |   movel([0.287883, -0.614127, -2.825456, -1.272806, 1.570796, 1.858679],accel_mss,speed_ms,0,blend_radius_m)
    |   movel([0.292066, -0.609849, -2.825809, -1.276731, 1.570796, 1.862863],accel_mss,speed_ms,0,blend_radius_m)
    |   movel([0.296239, -0.605302, -2.826176, -1.280911, 1.570796, 1.867035],accel_mss,speed_ms,0,blend_radius_m)
    |   movel([0.304565, -0.595657, -2.826929, -1.289803, 1.570796, 1.875361],accel_mss,speed_ms,0,blend_radius_m)
    |   movel([0.312884, -0.585713, -2.827668, -1.299008, 1.570796, 1.883680],accel_mss,speed_ms,0,blend_radius_m)
    |   movel([0.321462, -0.575765, -2.828370, -1.308254, 1.570796, 1.892259],accel_mss,speed_ms,0,blend_radius_m)
    |   movel([0.325905, -0.570907, -2.828700, -1.312783, 1.570796, 1.896702],accel_mss,speed_ms,0,blend_radius_m)
    |   movel([0.330404, -0.566266, -2.829006, -1.317117, 1.570796, 1.901200],accel_mss,speed_ms,0,blend_radius_m)
    |   movel([0.334923, -0.561932, -2.829285, -1.321171, 1.570796, 1.905719],accel_mss,speed_ms,0,blend_radius_m)
    |   movel([0.339422, -0.558022, -2.829531, -1.324836, 1.570796, 1.910218],accel_mss,speed_ms,0,blend_radius_m)
    |   movel([0.343854, -0.554640, -2.829740, -1.328010, 1.570796, 1.914650],accel_mss,speed_ms,0,blend_radius_m)
    |   movel([0.348182, -0.551894, -2.829906, -1.330589, 1.570796, 1.918978],accel_mss,speed_ms,0,blend_radius_m)
    |   movel([0.357075, -0.547601, -2.830160, -1.334628, 1.570796, 1.927872],accel_mss,speed_ms,0,blend_radius_m)
    |   movel([0.360141, -0.545901, -2.830259, -1.336229, 1.570796, 1.930937],accel_mss,speed_ms,0,blend_radius_m)
    |   movel([0.363459, -0.543566, -2.830393, -1.338430, 1.570796, 1.934255],accel_mss,speed_ms,0,blend_radius_m)
    |   movel([0.366887, -0.540552, -2.830563, -1.341275, 1.570796, 1.937683],accel_mss,speed_ms,0,blend_radius_m)
    |   movel([0.370117, -0.537011, -2.830758, -1.344620, 1.570796, 1.940913],accel_mss,speed_ms,0,blend_radius_m)
    |   movel([0.371567, -0.535082, -2.830863, -1.346444, 1.570796, 1.942363],accel_mss,speed_ms,0,blend_radius_m)
    |   movel([0.372854, -0.533077, -2.830971, -1.348342, 1.570796, 1.943650],accel_mss,speed_ms,0,blend_radius_m)
    |   speed_ms = 0.005
    |   movel([0.372854, -0.528532, -2.824043, -1.359814, 1.570796, 1.943650],accel_mss,speed_ms,0,blend_radius_m)
    |   speed_ms = 0.040
    |   movel([0.392993, -0.492142, -2.825739, -1.394509, 1.570796, 1.963790],accel_mss,speed_ms,0,blend_radius_m)
    |   speed_ms = 0.005
    |   movel([0.392993, -0.495981, -2.832703, -1.383705, 1.570796, 1.963790],accel_mss,speed_ms,0,blend_radius_m)
    |   speed_ms = 0.025
    |   movel([0.393910, -0.496024, -2.832701, -1.383664, 1.570796, 1.964707],accel_mss,speed_ms,0,blend_radius_m)
    |   movel([0.393756, -0.497351, -2.832647, -1.382391, 1.570796, 1.964553],accel_mss,speed_ms,0,blend_radius_m)
    |   movel([0.392785, -0.499332, -2.832566, -1.380491, 1.570796, 1.963582],accel_mss,speed_ms,0,blend_radius_m)
    |   movel([0.391276, -0.501335, -2.832482, -1.378572, 1.570796, 1.962072],accel_mss,speed_ms,0,blend_radius_m)
    |   movel([0.389590, -0.502920, -2.832415, -1.377054, 1.570796, 1.960387],accel_mss,speed_ms,0,blend_radius_m)
    |   movel([0.387923, -0.504170, -2.832362, -1.375857, 1.570796, 1.958719],accel_mss,speed_ms,0,blend_radius_m)
    |   movel([0.384630, -0.506318, -2.832268, -1.373802, 1.570796, 1.955427],accel_mss,speed_ms,0,blend_radius_m)
    |   movel([0.382205, -0.508147, -2.832188, -1.372055, 1.570796, 1.953002],accel_mss,speed_ms,0,blend_radius_m)
    |   movel([0.379769, -0.510289, -2.832092, -1.370008, 1.570796, 1.950565],accel_mss,speed_ms,0,blend_radius_m)
    |   movel([0.374902, -0.515289, -2.831861, -1.365239, 1.570796, 1.945699],accel_mss,speed_ms,0,blend_radius_m)
    |   movel([0.370138, -0.520881, -2.831593, -1.359915, 1.570796, 1.940935],accel_mss,speed_ms,0,blend_radius_m)
    |   movel([0.365584, -0.526607, -2.831308, -1.354475, 1.570796, 1.936381],accel_mss,speed_ms,0,blend_radius_m)
    |   movel([0.364539, -0.528025, -2.831235, -1.353129, 1.570796, 1.935335],accel_mss,speed_ms,0,blend_radius_m)
    |   movel([0.363843, -0.529356, -2.831166, -1.351867, 1.570796, 1.934639],accel_mss,speed_ms,0,blend_radius_m)
    |   movel([0.363932, -0.530295, -2.831117, -1.350977, 1.570796, 1.934728],accel_mss,speed_ms,0,blend_radius_m)
    |   movel([0.364709, -0.530522, -2.831105, -1.350761, 1.570796, 1.935505],accel_mss,speed_ms,0,blend_radius_m)
    |   movel([0.366882, -0.530324, -2.831116, -1.350949, 1.570796, 1.937678],accel_mss,speed_ms,0,blend_radius_m)
    |   movel([0.369349, -0.529593, -2.831154, -1.351642, 1.570796, 1.940145],accel_mss,speed_ms,0,blend_radius_m)
    |   movel([0.372065, -0.528370, -2.831217, -1.352802, 1.570796, 1.942862],accel_mss,speed_ms,0,blend_radius_m)
    |   movel([0.374984, -0.526670, -2.831304, -1.354414, 1.570796, 1.945780],accel_mss,speed_ms,0,blend_radius_m)
    |   movel([0.378038, -0.524551, -2.831411, -1.356427, 1.570796, 1.948835],accel_mss,speed_ms,0,blend_radius_m)
    |   movel([0.381188, -0.522022, -2.831537, -1.358830, 1.570796, 1.951985],accel_mss,speed_ms,0,blend_radius_m)
    |   movel([0.384371, -0.519133, -2.831678, -1.361578, 1.570796, 1.955167],accel_mss,speed_ms,0,blend_radius_m)
    |   movel([0.387541, -0.515900, -2.831833, -1.364656, 1.570796, 1.958338],accel_mss,speed_ms,0,blend_radius_m)
    |   movel([0.386816, -0.517857, -2.831740, -1.362792, 1.570796, 1.957612],accel_mss,speed_ms,0,blend_radius_m)
    |   movel([0.386885, -0.519218, -2.831674, -1.361497, 1.570796, 1.957682],accel_mss,speed_ms,0,blend_radius_m)
    |   movel([0.387619, -0.519910, -2.831641, -1.360838, 1.570796, 1.958415],accel_mss,speed_ms,0,blend_radius_m)
    |   movel([0.388878, -0.519866, -2.831643, -1.360881, 1.570796, 1.959674],accel_mss,speed_ms,0,blend_radius_m)
    |   movel([0.390482, -0.519148, -2.831678, -1.361564, 1.570796, 1.961278],accel_mss,speed_ms,0,blend_radius_m)
    |   movel([0.392279, -0.517965, -2.831734, -1.362689, 1.570796, 1.963075],accel_mss,speed_ms,0,blend_radius_m)
    |   movel([0.396102, -0.514741, -2.831887, -1.365761, 1.570796, 1.966899],accel_mss,speed_ms,0,blend_radius_m)
    |   movel([0.401023, -0.509879, -2.832110, -1.370400, 1.570796, 1.971819],accel_mss,speed_ms,0,blend_radius_m)
    |   movel([0.405829, -0.504489, -2.832348, -1.375552, 1.570796, 1.976625],accel_mss,speed_ms,0,blend_radius_m)
    |   movel([0.410389, -0.498733, -2.832591, -1.381066, 1.570796, 1.981185],accel_mss,speed_ms,0,blend_radius_m)
    |   movel([0.414565, -0.492767, -2.832830, -1.386792, 1.570796, 1.985361],accel_mss,speed_ms,0,blend_radius_m)
    |   movel([0.415797, -0.490746, -2.832908, -1.388734, 1.570796, 1.986593],accel_mss,speed_ms,0,blend_radius_m)
    |   movel([0.416474, -0.489006, -2.832975, -1.390408, 1.570796, 1.987270],accel_mss,speed_ms,0,blend_radius_m)
    |   movel([0.416317, -0.488122, -2.833008, -1.391259, 1.570796, 1.987113],accel_mss,speed_ms,0,blend_radius_m)
    |   movel([0.415708, -0.487718, -2.833023, -1.391647, 1.570796, 1.986505],accel_mss,speed_ms,0,blend_radius_m)
    |   movel([0.413037, -0.487241, -2.833041, -1.392107, 1.570796, 1.983833],accel_mss,speed_ms,0,blend_radius_m)
    |   movel([0.407478, -0.487250, -2.833041, -1.392098, 1.570796, 1.978275],accel_mss,speed_ms,0,blend_radius_m)
    |   movel([0.405255, -0.486145, -2.833082, -1.393163, 1.570796, 1.976051],accel_mss,speed_ms,0,blend_radius_m)
    |   movel([0.410957, -0.479463, -2.833320, -1.399605, 1.570796, 1.981754],accel_mss,speed_ms,0,blend_radius_m)
    |   movel([0.413948, -0.476450, -2.833423, -1.402516, 1.570796, 1.984745],accel_mss,speed_ms,0,blend_radius_m)
    |   movel([0.416947, -0.473850, -2.833509, -1.405030, 1.570796, 1.987743],accel_mss,speed_ms,0,blend_radius_m)
    |   movel([0.418941, -0.472429, -2.833555, -1.406405, 1.570796, 1.989737],accel_mss,speed_ms,0,blend_radius_m)
    |   movel([0.420949, -0.471263, -2.833592, -1.407534, 1.570796, 1.991746],accel_mss,speed_ms,0,blend_radius_m)
    |   movel([0.424362, -0.469990, -2.833632, -1.408766, 1.570796, 1.995159],accel_mss,speed_ms,0,blend_radius_m)
    |   movel([0.425900, -0.470389, -2.833620, -1.408380, 1.570796, 1.996696],accel_mss,speed_ms,0,blend_radius_m)
    |   movel([0.426184, -0.471160, -2.833595, -1.407634, 1.570796, 1.996980],accel_mss,speed_ms,0,blend_radius_m)
    |   movel([0.426032, -0.472341, -2.833558, -1.406491, 1.570796, 1.996829],accel_mss,speed_ms,0,blend_radius_m)
    |   movel([0.425184, -0.474318, -2.833493, -1.404577, 1.570796, 1.995980],accel_mss,speed_ms,0,blend_radius_m)
    |   movel([0.423811, -0.476494, -2.833421, -1.402474, 1.570796, 1.994607],accel_mss,speed_ms,0,blend_radius_m)
    |   movel([0.420302, -0.480879, -2.833271, -1.398239, 1.570796, 1.991098],accel_mss,speed_ms,0,blend_radius_m)
    |   speed_ms = 0.005
    |   movel([0.420302, -0.477335, -2.826295, -1.408760, 1.570796, 1.991098],accel_mss,speed_ms,0,blend_radius_m)
    |   speed_ms = 0.040
    |   movel([0.476664, -0.338700, -2.827888, -1.545801, 1.570796, 2.047460],accel_mss,speed_ms,0,blend_radius_m)
    |   speed_ms = 0.005
    |   movel([0.476664, -0.339316, -2.834899, -1.538174, 1.570796, 2.047460],accel_mss,speed_ms,0,blend_radius_m)
    |   speed_ms = 0.025
    |   movel([0.479370, -0.336834, -2.834869, -1.540686, 1.570796, 2.050166],accel_mss,speed_ms,0,blend_radius_m)
    |   movel([0.481986, -0.334757, -2.834843, -1.542789, 1.570796, 2.052782],accel_mss,speed_ms,0,blend_radius_m)
    |   movel([0.484460, -0.333094, -2.834821, -1.544475, 1.570796, 2.055256],accel_mss,speed_ms,0,blend_radius_m)
    |   movel([0.488820, -0.331033, -2.834792, -1.546564, 1.570796, 2.059617],accel_mss,speed_ms,0,blend_radius_m)
    |   movel([0.490616, -0.330643, -2.834786, -1.546960, 1.570796, 2.061412],accel_mss,speed_ms,0,blend_radius_m)
    |   movel([0.493217, -0.331170, -2.834794, -1.546426, 1.570796, 2.064013],accel_mss,speed_ms,0,blend_radius_m)
    |   movel([0.494459, -0.333234, -2.834823, -1.544332, 1.570796, 2.065255],accel_mss,speed_ms,0,blend_radius_m)
    |   movel([0.494608, -0.336421, -2.834864, -1.541104, 1.570796, 2.065405],accel_mss,speed_ms,0,blend_radius_m)
    |   movel([0.493895, -0.340430, -2.834912, -1.537047, 1.570796, 2.064691],accel_mss,speed_ms,0,blend_radius_m)
    |   movel([0.492547, -0.344965, -2.834960, -1.532464, 1.570796, 2.063343],accel_mss,speed_ms,0,blend_radius_m)
    |   movel([0.489670, -0.352434, -2.835024, -1.524931, 1.570796, 2.060466],accel_mss,speed_ms,0,blend_radius_m)
    |   movel([0.485945, -0.360458, -2.835073, -1.516859, 1.570796, 2.056741],accel_mss,speed_ms,0,blend_radius_m)
    |   movel([0.481457, -0.368888, -2.835102, -1.508400, 1.570796, 2.052253],accel_mss,speed_ms,0,blend_radius_m)
    |   movel([0.471336, -0.385808, -2.835090, -1.491491, 1.570796, 2.042132],accel_mss,speed_ms,0,blend_radius_m)
    |   movel([0.469595, -0.389450, -2.835075, -1.487865, 1.570796, 2.040391],accel_mss,speed_ms,0,blend_radius_m)
    |   movel([0.468924, -0.392314, -2.835060, -1.485015, 1.570796, 2.039720],accel_mss,speed_ms,0,blend_radius_m)
    |   movel([0.469444, -0.393862, -2.835051, -1.483476, 1.570796, 2.040240],accel_mss,speed_ms,0,blend_radius_m)
    |   movel([0.470629, -0.394698, -2.835046, -1.482645, 1.570796, 2.041425],accel_mss,speed_ms,0,blend_radius_m)
    |   movel([0.471949, -0.395400, -2.835041, -1.481948, 1.570796, 2.042746],accel_mss,speed_ms,0,blend_radius_m)
    |   movel([0.472859, -0.396556, -2.835034, -1.480799, 1.570796, 2.043656],accel_mss,speed_ms,0,blend_radius_m)
    |   movel([0.472981, -0.398305, -2.835021, -1.479063, 1.570796, 2.043778],accel_mss,speed_ms,0,blend_radius_m)
    |   movel([0.472503, -0.400598, -2.835003, -1.476788, 1.570796, 2.043300],accel_mss,speed_ms,0,blend_radius_m)
    |   movel([0.470523, -0.406016, -2.834953, -1.471420, 1.570796, 2.041320],accel_mss,speed_ms,0,blend_radius_m)
    |   movel([0.466993, -0.414215, -2.834860, -1.463315, 1.570796, 2.037789],accel_mss,speed_ms,0,blend_radius_m)
    |   movel([0.463094, -0.422600, -2.834741, -1.455048, 1.570796, 2.033890],accel_mss,speed_ms,0,blend_radius_m)
    |   movel([0.458842, -0.431131, -2.834597, -1.446661, 1.570796, 2.029638],accel_mss,speed_ms,0,blend_radius_m)
    |   movel([0.454272, -0.439773, -2.834426, -1.438190, 1.570796, 2.025068],accel_mss,speed_ms,0,blend_radius_m)
    |   movel([0.449406, -0.448477, -2.834229, -1.429684, 1.570796, 2.020203],accel_mss,speed_ms,0,blend_radius_m)
    |   movel([0.444281, -0.457203, -2.834006, -1.421181, 1.570796, 2.015077],accel_mss,speed_ms,0,blend_radius_m)
    |   movel([0.438899, -0.465925, -2.833757, -1.412707, 1.570796, 2.009695],accel_mss,speed_ms,0,blend_radius_m)
    |   movel([0.433294, -0.474608, -2.833484, -1.404297, 1.570796, 2.004091],accel_mss,speed_ms,0,blend_radius_m)
    |   movel([0.429578, -0.480057, -2.833300, -1.399033, 1.570796, 2.000375],accel_mss,speed_ms,0,blend_radius_m)
    |   movel([0.425574, -0.485395, -2.833109, -1.393884, 1.570796, 1.996371],accel_mss,speed_ms,0,blend_radius_m)
    |   movel([0.421375, -0.490220, -2.832929, -1.389241, 1.570796, 1.992172],accel_mss,speed_ms,0,blend_radius_m)
    |   movel([0.419234, -0.492302, -2.832848, -1.387239, 1.570796, 1.990031],accel_mss,speed_ms,0,blend_radius_m)
    |   movel([0.417072, -0.494113, -2.832777, -1.385499, 1.570796, 1.987868],accel_mss,speed_ms,0,blend_radius_m)
    |   speed_ms = 0.005
    |   movel([0.417072, -0.490310, -2.825811, -1.396267, 1.570796, 1.987868],accel_mss,speed_ms,0,blend_radius_m)
    |   speed_ms = 0.040
    |   movel([0.404965, -0.505233, -2.825183, -1.381973, 1.570796, 1.975761],accel_mss,speed_ms,0,blend_radius_m)
    |   speed_ms = 0.005
    |   movel([0.404965, -0.509329, -2.832135, -1.370925, 1.570796, 1.975761],accel_mss,speed_ms,0,blend_radius_m)
    |   speed_ms = 0.025
    |   movel([0.405117, -0.510451, -2.832084, -1.369854, 1.570796, 1.975914],accel_mss,speed_ms,0,blend_radius_m)
    |   movel([0.404551, -0.512177, -2.832006, -1.368206, 1.570796, 1.975347],accel_mss,speed_ms,0,blend_radius_m)
    |   movel([0.403457, -0.514211, -2.831912, -1.366266, 1.570796, 1.974254],accel_mss,speed_ms,0,blend_radius_m)
    |   movel([0.402012, -0.516256, -2.831816, -1.364317, 1.570796, 1.972809],accel_mss,speed_ms,0,blend_radius_m)
    |   movel([0.400072, -0.518346, -2.831716, -1.362327, 1.570796, 1.970868],accel_mss,speed_ms,0,blend_radius_m)
    |   movel([0.398135, -0.520018, -2.831635, -1.360736, 1.570796, 1.968931],accel_mss,speed_ms,0,blend_radius_m)
    |   movel([0.396249, -0.521587, -2.831559, -1.359244, 1.570796, 1.967045],accel_mss,speed_ms,0,blend_radius_m)
    |   movel([0.394483, -0.523364, -2.831471, -1.357555, 1.570796, 1.965279],accel_mss,speed_ms,0,blend_radius_m)
    |   movel([0.392507, -0.526332, -2.831321, -1.354735, 1.570796, 1.963303],accel_mss,speed_ms,0,blend_radius_m)
    |   movel([0.391580, -0.527872, -2.831243, -1.353274, 1.570796, 1.962377],accel_mss,speed_ms,0,blend_radius_m)
    |   movel([0.390374, -0.529514, -2.831158, -1.351717, 1.570796, 1.961170],accel_mss,speed_ms,0,blend_radius_m)
    |   movel([0.386716, -0.533607, -2.830942, -1.347840, 1.570796, 1.957512],accel_mss,speed_ms,0,blend_radius_m)
    |   movel([0.383094, -0.537143, -2.830751, -1.344495, 1.570796, 1.953891],accel_mss,speed_ms,0,blend_radius_m)
    |   movel([0.379475, -0.540207, -2.830582, -1.341600, 1.570796, 1.950271],accel_mss,speed_ms,0,blend_radius_m)
    |   movel([0.375819, -0.542917, -2.830430, -1.339043, 1.570796, 1.946615],accel_mss,speed_ms,0,blend_radius_m)
    |   movel([0.377746, -0.541315, -2.830520, -1.340554, 1.570796, 1.948542],accel_mss,speed_ms,0,blend_radius_m)
    |   movel([0.379610, -0.540015, -2.830593, -1.341781, 1.570796, 1.950407],accel_mss,speed_ms,0,blend_radius_m)
    |   movel([0.381213, -0.539414, -2.830626, -1.342349, 1.570796, 1.952009],accel_mss,speed_ms,0,blend_radius_m)
    |   movel([0.382103, -0.539913, -2.830598, -1.341877, 1.570796, 1.952899],accel_mss,speed_ms,0,blend_radius_m)
    |   movel([0.381891, -0.541549, -2.830507, -1.340333, 1.570796, 1.952687],accel_mss,speed_ms,0,blend_radius_m)
    |   movel([0.380839, -0.543723, -2.830384, -1.338282, 1.570796, 1.951635],accel_mss,speed_ms,0,blend_radius_m)
    |   movel([0.379288, -0.545943, -2.830256, -1.336190, 1.570796, 1.950084],accel_mss,speed_ms,0,blend_radius_m)
    |   movel([0.374627, -0.551255, -2.829944, -1.331190, 1.570796, 1.945423],accel_mss,speed_ms,0,blend_radius_m)
    |   movel([0.371659, -0.554205, -2.829766, -1.328418, 1.570796, 1.942455],accel_mss,speed_ms,0,blend_radius_m)
    |   movel([0.368690, -0.556856, -2.829604, -1.325929, 1.570796, 1.939487],accel_mss,speed_ms,0,blend_radius_m)
    |   movel([0.365749, -0.559177, -2.829459, -1.323752, 1.570796, 1.936545],accel_mss,speed_ms,0,blend_radius_m)
    |   movel([0.369015, -0.557012, -2.829594, -1.325782, 1.570796, 1.939811],accel_mss,speed_ms,0,blend_radius_m)
    |   movel([0.372492, -0.554335, -2.829758, -1.328296, 1.570796, 1.943288],accel_mss,speed_ms,0,blend_radius_m)
    |   movel([0.375890, -0.551784, -2.829912, -1.330692, 1.570796, 1.946686],accel_mss,speed_ms,0,blend_radius_m)
    |   movel([0.378923, -0.549976, -2.830020, -1.332393, 1.570796, 1.949719],accel_mss,speed_ms,0,blend_radius_m)
    |   movel([0.379701, -0.549871, -2.830026, -1.332492, 1.570796, 1.950497],accel_mss,speed_ms,0,blend_radius_m)
    |   movel([0.379616, -0.550533, -2.829987, -1.331869, 1.570796, 1.950413],accel_mss,speed_ms,0,blend_radius_m)
    |   movel([0.377499, -0.554136, -2.829770, -1.328483, 1.570796, 1.948296],accel_mss,speed_ms,0,blend_radius_m)
    |   movel([0.375650, -0.556761, -2.829610, -1.326018, 1.570796, 1.946446],accel_mss,speed_ms,0,blend_radius_m)
    |   movel([0.373642, -0.559288, -2.829452, -1.323648, 1.570796, 1.944438],accel_mss,speed_ms,0,blend_radius_m)
    |   movel([0.371528, -0.561649, -2.829303, -1.321437, 1.570796, 1.942324],accel_mss,speed_ms,0,blend_radius_m)
    |   movel([0.372560, -0.560724, -2.829362, -1.322303, 1.570796, 1.943356],accel_mss,speed_ms,0,blend_radius_m)
    |   movel([0.373665, -0.560011, -2.829407, -1.322971, 1.570796, 1.944462],accel_mss,speed_ms,0,blend_radius_m)
    |   movel([0.375965, -0.559172, -2.829460, -1.323758, 1.570796, 1.946762],accel_mss,speed_ms,0,blend_radius_m)
    |   movel([0.378139, -0.559065, -2.829466, -1.323858, 1.570796, 1.948935],accel_mss,speed_ms,0,blend_radius_m)
    |   movel([0.379917, -0.559608, -2.829432, -1.323348, 1.570796, 1.950714],accel_mss,speed_ms,0,blend_radius_m)
    |   movel([0.381037, -0.560714, -2.829363, -1.322312, 1.570796, 1.951833],accel_mss,speed_ms,0,blend_radius_m)
    |   movel([0.381236, -0.562286, -2.829263, -1.320840, 1.570796, 1.952032],accel_mss,speed_ms,0,blend_radius_m)
    |   movel([0.380909, -0.563217, -2.829203, -1.319968, 1.570796, 1.951705],accel_mss,speed_ms,0,blend_radius_m)
    |   movel([0.380254, -0.564226, -2.829139, -1.319024, 1.570796, 1.951050],accel_mss,speed_ms,0,blend_radius_m)
    |   movel([0.379243, -0.565312, -2.829068, -1.318009, 1.570796, 1.950040],accel_mss,speed_ms,0,blend_radius_m)
    |   movel([0.377837, -0.566454, -2.828994, -1.316941, 1.570796, 1.948633],accel_mss,speed_ms,0,blend_radius_m)
    |   movel([0.376345, -0.567293, -2.828939, -1.316157, 1.570796, 1.947141],accel_mss,speed_ms,0,blend_radius_m)
    |   movel([0.371088, -0.568361, -2.828869, -1.315159, 1.570796, 1.941884],accel_mss,speed_ms,0,blend_radius_m)
    |   movel([0.369018, -0.568917, -2.828832, -1.314640, 1.570796, 1.939814],accel_mss,speed_ms,0,blend_radius_m)
    |   movel([0.366727, -0.569974, -2.828762, -1.313653, 1.570796, 1.937523],accel_mss,speed_ms,0,blend_radius_m)
    |   movel([0.362562, -0.572897, -2.828566, -1.310927, 1.570796, 1.933358],accel_mss,speed_ms,0,blend_radius_m)
    |   movel([0.358323, -0.576137, -2.828344, -1.307908, 1.570796, 1.929119],accel_mss,speed_ms,0,blend_radius_m)
    |   movel([0.356263, -0.577399, -2.828257, -1.306732, 1.570796, 1.927059],accel_mss,speed_ms,0,blend_radius_m)
    |   movel([0.354408, -0.578139, -2.828206, -1.306044, 1.570796, 1.925204],accel_mss,speed_ms,0,blend_radius_m)
    |   movel([0.353007, -0.578145, -2.828205, -1.306038, 1.570796, 1.923804],accel_mss,speed_ms,0,blend_radius_m)
    |   movel([0.352301, -0.577219, -2.828270, -1.306901, 1.570796, 1.923097],accel_mss,speed_ms,0,blend_radius_m)
    |   movel([0.354575, -0.574223, -2.828476, -1.309691, 1.570796, 1.925371],accel_mss,speed_ms,0,blend_radius_m)
    |   movel([0.356998, -0.571354, -2.828670, -1.312366, 1.570796, 1.927794],accel_mss,speed_ms,0,blend_radius_m)
    |   speed_ms = 0.005
    |   movel([0.356998, -0.566113, -2.821791, -1.324485, 1.570796, 1.927794],accel_mss,speed_ms,0,blend_radius_m)
    |   speed_ms = 0.040
    |   movel([0.372981, -0.575681, -2.821133, -1.315575, 1.570796, 1.943777],accel_mss,speed_ms,0,blend_radius_m)
    |   speed_ms = 0.005
    |   movel([0.372981, -0.581093, -2.827999, -1.303297, 1.570796, 1.943777],accel_mss,speed_ms,0,blend_radius_m)
    |   speed_ms = 0.025
    |   movel([0.374590, -0.578956, -2.828149, -1.305284, 1.570796, 1.945386],accel_mss,speed_ms,0,blend_radius_m)
    |   movel([0.376451, -0.577299, -2.828264, -1.306825, 1.570796, 1.947247],accel_mss,speed_ms,0,blend_radius_m)
    |   movel([0.378267, -0.576269, -2.828335, -1.307784, 1.570796, 1.949063],accel_mss,speed_ms,0,blend_radius_m)
    |   movel([0.379725, -0.576023, -2.828352, -1.308014, 1.570796, 1.950522],accel_mss,speed_ms,0,blend_radius_m)
    |   movel([0.380680, -0.576510, -2.828319, -1.307560, 1.570796, 1.951476],accel_mss,speed_ms,0,blend_radius_m)
    |   movel([0.381263, -0.577469, -2.828252, -1.306668, 1.570796, 1.952059],accel_mss,speed_ms,0,blend_radius_m)
    |   movel([0.381788, -0.580128, -2.828067, -1.304194, 1.570796, 1.952584],accel_mss,speed_ms,0,blend_radius_m)
    |   movel([0.383315, -0.577532, -2.828248, -1.306609, 1.570796, 1.954112],accel_mss,speed_ms,0,blend_radius_m)
    |   movel([0.384367, -0.575051, -2.828419, -1.308919, 1.570796, 1.955164],accel_mss,speed_ms,0,blend_radius_m)
    |   movel([0.384857, -0.572901, -2.828565, -1.310922, 1.570796, 1.955654],accel_mss,speed_ms,0,blend_radius_m)
    |   movel([0.384731, -0.571259, -2.828676, -1.312454, 1.570796, 1.955527],accel_mss,speed_ms,0,blend_radius_m)
    |   movel([0.385607, -0.571687, -2.828647, -1.312055, 1.570796, 1.956403],accel_mss,speed_ms,0,blend_radius_m)
    |   movel([0.386172, -0.572484, -2.828594, -1.311311, 1.570796, 1.956969],accel_mss,speed_ms,0,blend_radius_m)
    |   movel([0.386545, -0.574933, -2.828427, -1.309029, 1.570796, 1.957342],accel_mss,speed_ms,0,blend_radius_m)
    |   movel([0.386215, -0.578123, -2.828207, -1.306059, 1.570796, 1.957011],accel_mss,speed_ms,0,blend_radius_m)
    |   movel([0.385505, -0.581607, -2.827962, -1.302820, 1.570796, 1.956301],accel_mss,speed_ms,0,blend_radius_m)
    |   movel([0.384235, -0.585688, -2.827670, -1.299032, 1.570796, 1.955031],accel_mss,speed_ms,0,blend_radius_m)
    |   movel([0.382537, -0.589777, -2.827370, -1.295241, 1.570796, 1.953334],accel_mss,speed_ms,0,blend_radius_m)
    |   movel([0.380801, -0.593813, -2.827069, -1.291508, 1.570796, 1.951597],accel_mss,speed_ms,0,blend_radius_m)
    |   movel([0.379403, -0.597748, -2.826769, -1.287873, 1.570796, 1.950199],accel_mss,speed_ms,0,blend_radius_m)
    |   movel([0.378430, -0.596064, -2.826898, -1.289427, 1.570796, 1.949227],accel_mss,speed_ms,0,blend_radius_m)
    |   movel([0.376831, -0.595184, -2.826965, -1.290241, 1.570796, 1.947628],accel_mss,speed_ms,0,blend_radius_m)
    |   movel([0.374646, -0.595186, -2.826965, -1.290238, 1.570796, 1.945442],accel_mss,speed_ms,0,blend_radius_m)
    |   movel([0.371905, -0.596154, -2.826891, -1.289344, 1.570796, 1.942702],accel_mss,speed_ms,0,blend_radius_m)
    |   speed_ms = 0.005
    |   movel([0.371905, -0.590481, -2.820049, -1.301859, 1.570796, 1.942702],accel_mss,speed_ms,0,blend_radius_m)
    |   speed_ms = 0.040
    |   movel([0.372964, -0.600587, -2.819260, -1.292543, 1.570796, 1.943761],accel_mss,speed_ms,0,blend_radius_m)
    |   speed_ms = 0.005
    |   movel([0.372964, -0.606434, -2.826085, -1.279870, 1.570796, 1.943761],accel_mss,speed_ms,0,blend_radius_m)
    |   speed_ms = 0.025
    |   movel([0.372672, -0.610833, -2.825728, -1.275827, 1.570796, 1.943468],accel_mss,speed_ms,0,blend_radius_m)
    |   movel([0.373070, -0.614605, -2.825416, -1.272367, 1.570796, 1.943866],accel_mss,speed_ms,0,blend_radius_m)
    |   movel([0.374414, -0.617284, -2.825191, -1.269914, 1.570796, 1.945211],accel_mss,speed_ms,0,blend_radius_m)
    |   movel([0.375527, -0.618067, -2.825125, -1.269197, 1.570796, 1.946323],accel_mss,speed_ms,0,blend_radius_m)
    |   movel([0.376979, -0.618403, -2.825096, -1.268889, 1.570796, 1.947775],accel_mss,speed_ms,0,blend_radius_m)
    |   movel([0.379455, -0.618070, -2.825125, -1.269194, 1.570796, 1.950251],accel_mss,speed_ms,0,blend_radius_m)
    |   movel([0.382276, -0.616958, -2.825219, -1.270212, 1.570796, 1.953072],accel_mss,speed_ms,0,blend_radius_m)
    |   movel([0.385374, -0.615245, -2.825363, -1.271781, 1.570796, 1.956170],accel_mss,speed_ms,0,blend_radius_m)
    |   movel([0.388671, -0.613110, -2.825541, -1.273739, 1.570796, 1.959467],accel_mss,speed_ms,0,blend_radius_m)
    |   movel([0.395561, -0.608282, -2.825936, -1.278171, 1.570796, 1.966357],accel_mss,speed_ms,0,blend_radius_m)
